(* CODESYS project xlh_palletizer_00_01.project
   Description: Receives some incoming messages and echoes them with CAN-ID +1
   Company: 3S - Smart Software Solutions GmbH
   Version: 1.0.0.0
   Title: CAN Bus API Example
   Author: 3S - Smart Software Solutions GmbH

Project tree, tasks and I/O mapping:
  xLH : CODESYS Control for Raspberry Pi 64 SL, CODESYS, order no. 2302000009, version 4.15.0.0
    application app
      libraries: Standard, 3.5.22.0 (System); Util, 3.5.22.0 (System); VisuDialogs, * (System); Memory, * (3S - Smart Software Solutions GmbH); xemax, 0.27 (xemax ag); CAN API, 1.0.0.4 (CODESYS)
      task MAIN_TASK (cyclic, interval 5 ms, priority 0) calls IO_READ, MAIN, MC, IO_WRITE
      task VISU_TASK (cyclic, interval 100 ms, priority 31) calls VisuElems.Visu_Prg
      task SoftMotion_PlanningTask (freewheeling, priority 15) calls nothing
      Symbols
      program MAIN [ST]
      visualisation Visualization
      MOTION/
        program MC [ST]: axSmExecuteToFalse, axGexecuteToFalse, axGenable, axGdisable, ipoGantry3
        trace PosControllerX (task MAIN_TASK): a1_axis.out.diSetVelocity, a1_axis.fSetAcceleration, a1_axis.fActPosition, a1_axis.fSetPosition, a1_axis.out.diSetVelocity
        function block FB_AXG_MOVE_ABSOLUTE [ST]
        function block FB_AXG_MOVE_RELATIVE [ST]
        trace PosController_A1_A2 (task MAIN_TASK): a1_axis.fSetPosition, a1_axis.fActPosition, a2_axis.fSetPosition, a2_axis.fActPosition
      IO/
        program IO_READ [ST]
        program io [ST]
        program IO_WRITE [ST]
      axis group AxisGroup: TRAFO.Kin_Gantry3, axes x_virtual, y_virtual, z_virtual
      text DemoInterpolator
      CNC settings
      text DemoXemaxLogo
      visualisation Visualization_1
      DOCS/
        Soft_Motion_Uebung_1_01_00
    SoftMotion General Axis Pool
      a3_axis : SM_Drive_PosControl, CODESYS, order no. 1805, version 4.18.0.0
          settings: wDriveID = 3; dwRatioTechUnitsDenom = 101846; iRatioTechUnitsNum = -125; eRampType = 0; fSWMaxAcceleration = 100; fSWMaxDeceleration = 100; fSWMaxJerk = 1000; fSWLimitNegative = -1000.0; ScalingIncs = 814768; ScalingUnits = 1000; InvertDirection = TRUE; IsLinearMotor = TRUE; MaximumOutputVelocityInt = 40738; MinimumOutputVelocityInt = -40738; Kp = 0.05; MaxFollowingError = 5.0; EnableFollowingErrorCheck = TRUE; DeadTime = 3.0
      a1_axis : SM_Drive_PosControl, CODESYS, order no. 1805, version 4.18.0.0
          settings: dwRatioTechUnitsDenom = 101846; iRatioTechUnitsNum = 125; eRampType = 0; fSWMaxVelocity = 50; fSWMaxAcceleration = 100; fSWMaxDeceleration = 100; fSWMaxJerk = 1000; fSWLimitNegative = -1000.0; ScalingIncs = 814768; ScalingUnits = 1000; IsLinearMotor = TRUE; MaximumOutputVelocityInt = 40738; MinimumOutputVelocityInt = -40738; Kp = 0.05; MaxFollowingError = 5.0; EnableFollowingErrorCheck = TRUE; DeadTime = 3.0
      a2_axis : SM_Drive_PosControl, CODESYS, order no. 1805, version 4.18.0.0
          settings: wDriveID = 2; dwRatioTechUnitsDenom = 101846; iRatioTechUnitsNum = 125; eRampType = 0; fSWMaxVelocity = 50; fSWMaxAcceleration = 100; fSWMaxDeceleration = 100; fSWMaxJerk = 1000; fSWLimitNegative = -1000.0; ScalingIncs = 814768; ScalingUnits = 1000; IsLinearMotor = TRUE; MaximumOutputVelocityInt = 40738; MinimumOutputVelocityInt = -40738; Kp = 0.05; MaxFollowingError = 5.0; EnableFollowingErrorCheck = TRUE; DeadTime = 3.0
      x_virtual : SM_Drive_Virtual, CODESYS, order no. 1805, version 4.18.0.0
          settings: wDriveID = 5; eRampType = 0; fSWMaxVelocity = 25; fSWMaxAcceleration = 100; fSWMaxDeceleration = 100; fSWMaxJerk = 1000; fSWLimitNegative = -1000.0
      y_virtual : SM_Drive_Virtual, CODESYS, order no. 1805, version 4.18.0.0
          settings: wDriveID = 6; eRampType = 0; fSWMaxVelocity = 25; fSWMaxAcceleration = 100; fSWMaxDeceleration = 100; fSWMaxJerk = 1000; fSWLimitNegative = -1000.0
      a4_axis : SM_Drive_PosControl, CODESYS, order no. 1805, version 4.18.0.0
          settings: wDriveID = 4; dwRatioTechUnitsDenom = 101846; iRatioTechUnitsNum = -125; eRampType = 0; fSWMaxAcceleration = 100; fSWMaxDeceleration = 100; fSWMaxJerk = 1000; fSWLimitNegative = -1000.0; ScalingIncs = 814768; ScalingUnits = 1000; InvertDirection = TRUE; IsLinearMotor = TRUE; MaximumOutputVelocityInt = 40738; MinimumOutputVelocityInt = -40738; Kp = 0.05; MaxFollowingError = 5.0; EnableFollowingErrorCheck = TRUE; DeadTime = 3.0
      z_virtual : SM_Drive_Virtual, CODESYS, order no. 1805, version 4.18.0.0
          settings: wDriveID = 7; eRampType = 0; fSWMaxVelocity = 25; fSWMaxAcceleration = 100; fSWMaxDeceleration = 100; fSWMaxJerk = 1000; fSWLimitNegative = -1000.0
    GPIOs_A_B : GPIOs B+/Pi2, CODESYS, version 4.15.0.0
        input  app.io.gpio.bSw1 : BOOL  // digital inputs (GPIO0..GPIO31).Bit4
        input  app.io.gpio.bSw2 : BOOL  // digital inputs (GPIO0..GPIO31).Bit5
        input  app.io.gpio.bSw3 : BOOL  // digital inputs (GPIO0..GPIO31).Bit6
        input  app.io.gpio.bSw4 : BOOL  // digital inputs (GPIO0..GPIO31).Bit12
        input  app.io.gpio.bSw5 : BOOL  // digital inputs (GPIO0..GPIO31).Bit13
        input  app.io.gpio.bSw6 : BOOL  // digital inputs (GPIO0..GPIO31).Bit16
        input  app.io.gpio.bSw7 : BOOL  // digital inputs (GPIO0..GPIO31).Bit17
        input  app.io.gpio.bSw8 : BOOL  // digital inputs (GPIO0..GPIO31).Bit19
        output app.io.gpio.bLed1 : BOOL  // digital outputs (GPIO0..GPIO31).Bit20
        output app.io.gpio.bLed2 : BOOL  // digital outputs (GPIO0..GPIO31).Bit21
        output app.io.gpio.bLed3 : BOOL  // digital outputs (GPIO0..GPIO31).Bit22
        output app.io.gpio.bLed4 : BOOL  // digital outputs (GPIO0..GPIO31).Bit23
        output app.io.gpio.bLed5 : BOOL  // digital outputs (GPIO0..GPIO31).Bit24
        output app.io.gpio.bLed6 : BOOL  // digital outputs (GPIO0..GPIO31).Bit26
        output app.io.gpio.bLed7 : BOOL  // digital outputs (GPIO0..GPIO31).Bit27
        unmapped channels: digital inputs (GPIO0..GPIO31), digital outputs (GPIO0..GPIO31)
    Onewire
    Camera device
      <Leer>
    SPI
    I²C
  libraries: VisuSymbols, 4.5.0.0 (System); DepictorBase, 1.2.0.0 (CODESYS)
  text list GlobalTextList
  00000000-0000-0000-0000-000000000000|E:\xemax ag\prj_24_03_xLH - Allgemein\Applikation\xLH_MOTION\CODESYS\Divers\080_SOFT_MOTION_PLC_OPEN\Soft_Motion_Uebung_1_01_00.pdf
*)

// xLH/app/IO/IO_READ
PROGRAM IO_READ
VAR
END_VAR

xemax.CAN_DRIVER();
io();
xemax.TASK_INFO();
xemax.LOCAL_TIME_AND_TIME_ZONE();

END_PROGRAM

// xLH/app/IO/io
PROGRAM io 
VAR_INPUT
	gpio: xemax.FB_XLH_GPIO;	
	motion: FB_XLH_MOTION := (uiCanIdBase:=16#300);
	xbox: FB_XBOX;
	bPenDown: BOOL;
END_VAR
VAR	
	bStartup: BOOL := TRUE;
	wdt: xemax.FB_XLH_WDT := (uiCanIdBase:=16#80);
	fbTonMagnet: TON;
END_VAR

IF bStartup THEN
	bStartup := FALSE;
	motion.pfbXlhMotionAxis[1] := ADR(MC.fbXlhMotionAxisA12.fbXlhMotionAxis1);
	motion.pfbXlhMotionAxis[2] := ADR(MC.fbXlhMotionAxisA12.fbXlhMotionAxis2);
	
	motion.uiIoOutPwmServo[9]  := 1000;
	
	CAN_DRIVER.mAddXlhDevice(pFbXlhIoDevice:=ADR(wdt));
	CAN_DRIVER.mAddXlhDevice(pFbXlhIoDevice:=ADR(motion));	
END_IF

xbox();

(*
IF io.bPenDown OR (z_virtual.fActPosition < (-1.0)) THEN
	motion.uiIoOutPwmServo[9]  := 1200;
ELSE
	motion.uiIoOutPwmServo[9]  := 800;
END_IF
*)

IF MC.iState < 3000 THEN
	IF bPenDown THEN
		motion.uiIoOutPwmServo[9]  := 1200;
	ELSE
		motion.uiIoOutPwmServo[9]  := 800;
	END_IF
ELSE
	IF z_virtual.fActPosition < (-1.0) THEN
		motion.uiIoOutPwmServo[9]  := 1200;
	ELSE
		motion.uiIoOutPwmServo[9]  := 800;
	END_IF
END_IF

END_PROGRAM

// xLH/app/MOTION/MC
PROGRAM MC
VAR_OUTPUT
	iState: INT;	
END_VAR
VAR
	bStartup: BOOL := TRUE;
	fbBlink: BLINK;
	
	axA1: FB_PLC_OPEN_AXIS := (rVel:=VEL, rAcc:=ACC_DEC, rDec:=ACC_DEC, rJerk:=JRK);
	axA2: FB_PLC_OPEN_AXIS := (rVel:=VEL, rAcc:=ACC_DEC, rDec:=ACC_DEC, rJerk:=JRK);
	axVx: FB_PLC_OPEN_AXIS := (rVel:=VEL, rAcc:=ACC_DEC, rDec:=ACC_DEC, rJerk:=JRK);
	axVy: FB_PLC_OPEN_AXIS := (rVel:=VEL, rAcc:=ACC_DEC, rDec:=ACC_DEC, rJerk:=JRK);
	axVz: FB_PLC_OPEN_AXIS := (rVel:=VEL, rAcc:=ACC_DEC, rDec:=ACC_DEC, rJerk:=JRK);
	fbXlhMotionAxisA12: FB_XLH_MOTION_AXIS_MID_T_BOT;
	fbTonDelay1: TON := (PT := TIME#1S0MS);
	fbTonDelay2: TON := (PT := TIME#1S0MS);	
	
	mcAxGenable : MC_GroupEnable;
	mcAxGdisable : MC_GroupDisable;
	mcAxGreset: MC_GroupReset;
	mcAxGsetCoord : MC_SetCoordinateTransform;	
	mcAxGmla: MC_MoveLinearAbsolute := (Velocity := VEL, Acceleration := ACC_DEC, Deceleration := ACC_DEC, Jerk := JRK);
	mcAxGmlr: MC_MoveLinearRelative := (Velocity := VEL, Acceleration := ACC_DEC, Deceleration := ACC_DEC, Jerk := JRK);	
	mcAxGcoordRef : MC_COORD_REF;
	smcPosRef: SMC_POS_REF;
	
	fbAxGmr: FB_AXG_MOVE_RELATIVE;
	fbAxGma: FB_AXG_MOVE_ABSOLUTE;
	
	rStepDistance: REAL := 15.0;
	rStpNeg: REAL;
	rStpPos: REAL;
	
	tPosMC : SMC_POS_REF ;
	smcGroupReadSetPosition : SMC_GroupReadSetPosition := (Enable:= TRUE, CoordSystem:= SMC_COORD_SYSTEM.MCS) ;
	mcGroupReadStatus: MC_GroupReadStatus;
	
	smcControlAxByPosA1: SMC_ControlAxisByPos;
	smcControlAxByPosA2: SMC_ControlAxisByPos;

	smcTrafoGantry3d: SMC_TRAFO_Gantry3;
	smcTrafofGantry3d: SMC_TRAFOF_Gantry3D;
	smcControlAxByPosX,smcControlAxByPosY, smcControlAxByPosZ: SMC_ControlAxisByPos;
	smcInterpolator: SMC_Interpolator;
	
	rOffsetX: REAL := 0.0;
	rOffsetY: REAL := -10.0;
	
	bVisuXplus: BOOL;
	bVisuXminus: BOOL;
	bVisuYplus: BOOL;
	bVisuYminus: BOOL;
	bVisuPenDown: BOOL;
	bVisuStartNc: BOOL;
	bVisuHoming: BOOL;
	
END_VAR
VAR CONSTANT
	VEL : REAL := 15.0;
	VEL_HOMING : REAL := 2.0;
    ACC_DEC : REAL := 100.0;
    JRK : REAL := 1000.0;	
END_VAR
VAR // added by the converter: edge detectors and wires of the graphical bodies
    _w1 : ANY;
END_VAR

// ToDo: Optimierung
IF bStartup THEN
	bStartup := FALSE;
	axA1.pAxis := ADR(a1_axis);
	axA2.pAxis := ADR(a2_axis);
	axVx.pAxis := ADR(x_virtual);
	axVy.pAxis := ADR(y_virtual);
	axVz.pAxis := ADR(z_virtual);
	
	fbXlhMotionAxisA12.fbXlhMotionAxis1.pAxis := ADR(a1_axis);
	fbXlhMotionAxisA12.fbXlhMotionAxis2.pAxis := ADR(a2_axis);
	fbXlhMotionAxisA12.pfbAxisPlcOpenX := ADR(axVx);
	fbXlhMotionAxisA12.pfbAxisPlcOpenY := ADR(axVy);
	fbXlhMotionAxisA12.pbEsX := ADR(io.motion.bIoIn[5]);
	fbXlhMotionAxisA12.pbEsY := ADR(io.motion.bIoIn[1]);
	
	fbAxGmr.axGmr REF= mcAxGmlr;
	fbAxGmr.axG REF= AxisGroup;  
	fbAxGma.axGma REF= mcAxGmla;
	fbAxGma.axG REF= AxisGroup;
	fbAxGma.axG REF= AxisGroup;
END_IF

axA1();
axA2();
fbXlhMotionAxisA12();
axVx();
axVy();
axVz();
MC.ipoGantry3();

// ToDo: Optimierung
mcAxGmla(AxisGroup:= AxisGroup);
mcAxGmlr(AxisGroup:= AxisGroup);
fbAxGmr();
fbAxGma();
mcGroupReadStatus(Enable:=TRUE, AxisGroup:=AxisGroup);
smcGroupReadSetPosition(Enable:=TRUE, AxisGroup:=AxisGroup, Position=>tPosMC);

tPosMC.c.X;
tPosMC.c.Y;
tPosMC.c.Z;
tPosMC.c.A;
tPosMC.c.B;
tPosMC.c.C;
a1_axis.fActPosition;
a2_axis.fActPosition;
x_virtual.fActPosition;
y_virtual.fActPosition;
z_virtual.fActPosition;

// kinematische Transformation
smcControlAxByPosA1(Axis:=a1_axis,
	        bEnable:= (iState >= 100),
            iStatus:=IPO_WAIT,
		    fSetPosition:= (+2.0) * x_virtual.fSetPosition + (+1.0) * y_virtual.fSetPosition,
			fGapVelocity:=VEL,
            fGapAcceleration:=ACC_DEC,
            fGapDeceleration:=ACC_DEC);
smcControlAxByPosA2(Axis:=a2_axis,
	        bEnable:= (iState >= 100),
            iStatus:=IPO_WAIT,
		    fSetPosition:= (+2.0) * x_virtual.fSetPosition - (+1.0) * y_virtual.fSetPosition,
			fGapVelocity:=VEL,
            fGapAcceleration:=ACC_DEC,
            fGapDeceleration:=ACC_DEC);

CASE iState OF
	// ============================================================================================
	// STARTUP UND INITIALISIERUNG
	// ============================================================================================
	
	0:		// Startup
			MC.axSmExecuteToFalse();
			MC.axGexecuteToFalse();		
			iState := 50;
			
	50:	// Power der Achsen
			axA1.mcp.Enable := TRUE; axA1.mcp.bRegulatorOn := TRUE; axA1.mcp.bDriveStart := TRUE;
			axA2.mcp.Enable := TRUE; axA2.mcp.bRegulatorOn := TRUE; axA2.mcp.bDriveStart := TRUE;
			// https://content.helpme-codesys.com/en/libs/SM3_Basic/Current/SM3_Basic/DataTypes/DriveInterface/SMC_AXIS_STATE.html
			IF (axA1.mcp.Status AND a1_axis.nAxisState = SMC_AXIS_STATE.standstill) AND
	           (axA2.mcp.Status AND a2_axis.nAxisState = SMC_AXIS_STATE.standstill) THEN
				MC.axSmExecuteToFalse();
				iState := iState + 10;
			END_IF
			
	60: // Power der Achsen
		axVx.mcp.Enable := TRUE; axVx.mcp.bRegulatorOn := TRUE; axVx.mcp.bDriveStart := TRUE;
		axVy.mcp.Enable := TRUE; axVy.mcp.bRegulatorOn := TRUE; axVy.mcp.bDriveStart := TRUE;
		axVz.mcp.Enable := TRUE; axVz.mcp.bRegulatorOn := TRUE; axVz.mcp.bDriveStart := TRUE;
		// https://content.helpme-codesys.com/en/libs/SM3_Basic/Current/SM3_Basic/DataTypes/DriveInterface/SMC_AXIS_STATE.html
		IF (axVx.mcp.Status AND x_virtual.nAxisState = SMC_AXIS_STATE.standstill) AND
		   (axVy.mcp.Status AND y_virtual.nAxisState = SMC_AXIS_STATE.standstill) AND
           (axVz.mcp.Status AND z_virtual.nAxisState = SMC_AXIS_STATE.standstill) THEN
			MC.axSmExecuteToFalse();
			iState := iState + 10;
		END_IF
		
	70: 	iState := 100;

	100:	// Disable der Achsengruppe		
			IF NOT mcGroupReadStatus.GroupDisabled THEN
				mcAxGdisable(AxisGroup := AxisGroup, Execute := TRUE);	
				IF mcAxGdisable.Done THEN
					MC.axGexecuteToFalse();
					iState := iState + 10;
				END_IF
			ELSE
				iState := iState + 10;
			END_IF	
			
	//110:	iState := iState + 20;

	110:	// Homing
			fbXlhMotionAxisA12.bHoming := TRUE;
			fbXlhMotionAxisA12.rVelHoming := VEL_HOMING;
			fbXlhMotionAxisA12.rVelHomingFast := 5.0 * VEL_HOMING;
			fbXlhMotionAxisA12.rOffsetX := 38.0;
			fbXlhMotionAxisA12.rOffsetY := -40.0;
			
			axVz.mcma.Execute := TRUE;
			axVz.mcma.Position := 0.0;
			axVz.mcma.Velocity := z_virtual.fSWMaxVelocity;
			
			IF fbXlhMotionAxisA12.bHomingDone AND
               axVz.mcma.Done THEN
				MC.axSmExecuteToFalse();
				fbXlhMotionAxisA12.bHoming := FALSE;
				iState := iState + 10;
			END_IF	
		
	120: 	iState := 1000;
	
	// ============================================================================================
	// Kommandos
	// ============================================================================================
	
	1000: 	// Resetierung der Kommandos
			MC.axSmExecuteToFalse();
			MC.axGexecuteToFalse();		
			
			bVisuXplus := FALSE;
			bVisuXminus := FALSE;
			bVisuYplus := FALSE;
			bVisuYminus := FALSE;
			//bVisuPenDown := FALSE;
			bVisuStartNc := FALSE;
			bVisuHoming := FALSE;
			
			iState := iState + 10;
			
	1010:	// warte auf Aktion					
			IF io.xbox.bRtBtnRightShoulder OR bVisuHoming THEN iState := 100; END_IF
						
			rStpNeg := rStepDistance * (-1.0);
			rStpPos := rStepDistance;
			
			IF io.xbox.bBtnB OR bVisuXplus    THEN smcPosRef.c.X := rStpPos; smcPosRef.c.Y := 0.0;	    iState := 2000; END_IF
			IF io.xbox.bBtnX OR bVisuXminus   THEN smcPosRef.c.X := rStpNeg; smcPosRef.c.Y := 0.0;	    iState := 2000; END_IF
			IF io.xbox.bBtnY OR bVisuYplus    THEN smcPosRef.c.X := 0.0;     smcPosRef.c.Y := rStpPos;	iState := 2000; END_IF
			IF io.xbox.bBtnA OR bVisuYminus   THEN smcPosRef.c.X := 0.0;     smcPosRef.c.Y := rStpNeg;	iState := 2000; END_IF
					
			//IF io.xbox.bBtnDpadUp   THEN io.bPenDown := FALSE; END_IF
			//IF io.xbox.bBtnDpadDown THEN io.bPenDown := TRUE;  END_IF
			io.bPenDown := bVisuPenDown;

			IF io.xbox.bBtnStart OR bVisuStartNc THEN iState := 3000; END_IF  
			
	// ============================================================================================
	// Stepbetrieb der Achsen
	// ============================================================================================
	
	// ToDo: Optimierung und Abstrahierung als FB
	
	
	2000:	MC.axGenable();
	2001: 	smcPosRef.c.Z := 0.0;
			fbAxGmr.bExecute := TRUE;
			fbAxGmr.tPosRef := smcPosRef;
			IF fbAxGmr.bDone THEN
				MC.axGexecuteToFalse();
				iState := iState + 1;
			END_IF
	2002:	MC.axGdisable();
	2003:	iState := 1000;
	
	2010:	MC.axGenable();
	2011: 	smcPosRef.c.Z := tPosMC.c.Z;
			fbAxGma.bExecute := TRUE;
			fbAxGma.tPosRef := smcPosRef;
			IF fbAxGma.bDone THEN
				MC.axGexecuteToFalse();
				iState := 1000;
			END_IF
	2012:	MC.axGdisable();
	2013:	iState := 1000;
			
	
	(*		
	2020: 	// Stifthalterung 
			smcPosRef.c.X := tPosMC.c.X;
			smcPosRef.c.Y := tPosMC.c.Y;
			IF io.bPenDown THEN
				smcPosRef.c.Z := -10.0;
			ELSE
				smcPosRef.c.Z := 0.0;
			END_IF
			fbAxGma.bExecute := TRUE;
			fbAxGma.tPosRef := smcPosRef;
			IF fbAxGma.bDone THEN
				MC.axGexecuteToFalse();
				iState := 1000;
			END_IF
	*)
	
	// ============================================================================================
	// Interpolator
	// ============================================================================================
	
	3000:	bVisuPenDown := FALSE;
			axVx.mcma.Execute := TRUE;
			axVx.mcma.Position := rOffsetX;
			axVy.mcma.Execute := TRUE;
			axVy.mcma.Position := rOffsetY;
			axVz.mcma.Execute := TRUE;
			axVz.mcma.Position := 0.0;
			IF axVx.mcma.Done AND axVy.mcma.Done AND axVz.mcma.Done THEN
				MC.axSmExecuteToFalse();
				iState := iState + 10;
			END_IF
			
	3010:	smcInterpolator.bExecute := TRUE;
			IF smcInterpolator.bDone THEN
				MC.axSmExecuteToFalse();
				iState := iState + 10;
			END_IF
			
	3020:	axVx.mcma.Execute := TRUE;
			axVx.mcma.Position := 0.0;
			axVy.mcma.Execute := TRUE;
			axVy.mcma.Position := 0.0;
			axVz.mcma.Execute := TRUE;
			axVz.mcma.Position := 0.0;
			IF axVx.mcma.Done AND axVy.mcma.Done AND axVz.mcma.Done THEN
				MC.axSmExecuteToFalse();
				iState := iState + 10;
			END_IF
	
	3030: 	iState := 1000;
	
	
END_CASE

fbTonDelay1();
fbTonDelay2();
fbTonDelay1.IN := FALSE;
fbTonDelay2.IN := FALSE;

ACTION axSmExecuteToFalse:
axA1.executeToFalse();
axA2.executeToFalse();
axVx.executeToFalse();
axVy.executeToFalse();
axVz.executeToFalse();

smcInterpolator.bExecute := FALSE;
END_ACTION

ACTION axGexecuteToFalse:
mcAxGenable(AxisGroup := AxisGroup, Execute := FALSE);
mcAxGdisable(AxisGroup := AxisGroup, Execute := FALSE);
mcAxGreset(AxisGroup := AxisGroup, Execute := FALSE);
mcAxGsetCoord(AxisGroup := AxisGroup, Execute := FALSE);

fbAxGma.bExecute := FALSE;
fbAxGmr.bExecute := FALSE;
mcAxGmla(AxisGroup := AxisGroup, Execute := FALSE);
mcAxGmlr(AxisGroup := AxisGroup, Execute := FALSE);
END_ACTION

ACTION axGenable:
// Enable der Achsengruppe
IF mcGroupReadStatus.GroupDisabled THEN 
	mcAxGenable(AxisGroup := AxisGroup, Execute := TRUE);	
	IF mcAxGenable.Done THEN
		MC.axGexecuteToFalse();
		iState := iState + 1;
		//iState := 580;
	END_IF			
END_IF	

// ToDo: Verallgemeinerung und Auslagerung in FB
END_ACTION

ACTION axGdisable:
// Disable der Achsengruppe		
IF NOT mcGroupReadStatus.GroupDisabled THEN
	mcAxGdisable(AxisGroup := AxisGroup, Execute := TRUE);	
	IF mcAxGdisable.Done THEN
		MC.axGexecuteToFalse();
		iState := iState + 1;
	END_IF
END_IF

// ToDo: Verallgemeinerung und Auslagerung in FB
END_ACTION

ACTION ipoGantry3:
smcTrafofGantry3d(
    minX := -50.0,
    maxX := 50.0,
    minY := -50.0,
    maxY := 50.0,
    minZ := -10.0,
    maxZ := 0.0,
    DriveX := x_virtual,
    DriveY := y_virtual,
    DriveZ := z_virtual); // SMC_TRAFOF_Gantry3D
smcControlAxByPosX(
    iStatus := smcInterpolator.iStatus,
    bEnable := smcInterpolator.bWorking,
    fSetPosition := smcTrafoGantry3d.dx,
    fGapVelocity := 10.0,
    fGapAcceleration := 100.0,
    fGapDeceleration := 100.0,
    Axis := x_virtual); // SMC_ControlAxisByPos
smcInterpolator(poqDataIn := ADR(DemoInterpolator), bEmergency_Stop := _w1, dwIpoTime := 5000); // SMC_Interpolator
smcTrafoGantry3d(pi := smcInterpolator.piSetPosition, dOffsetX := rOffsetX, dOffsetY := rOffsetY); // SMC_TRAFO_Gantry3
smcControlAxByPosY(
    iStatus := smcInterpolator.iStatus,
    bEnable := smcInterpolator.bWorking,
    fSetPosition := smcTrafoGantry3d.dy,
    fGapVelocity := 10.0,
    fGapAcceleration := 100.0,
    fGapDeceleration := 100.0,
    Axis := y_virtual); // SMC_ControlAxisByPos
smcControlAxByPosZ(
    iStatus := smcInterpolator.iStatus,
    bEnable := smcInterpolator.bWorking,
    fSetPosition := smcTrafoGantry3d.dz,
    fGapVelocity := 10.0,
    fGapAcceleration := 100.0,
    fGapDeceleration := 100.0,
    Axis := z_virtual); // SMC_ControlAxisByPos
_w1 := smcControlAxByPosX.bError OR smcControlAxByPosX.bStopIpo OR smcControlAxByPosY.bError OR smcControlAxByPosY.bStopIpo OR smcControlAxByPosZ.bError OR smcControlAxByPosZ.bStopIpo;
END_ACTION

END_PROGRAM

// xLH/app/MOTION/FB_AXG_MOVE_RELATIVE
FUNCTION_BLOCK FB_AXG_MOVE_RELATIVE
VAR_INPUT
	bExecute: BOOL;
	tPosRef: SMC_POS_REF;
	axGmr: REFERENCE TO MC_MoveLinearRelative;
	axG: REFERENCE TO AXIS_GROUP_REF_SM3;
END_VAR
VAR_OUTPUT
	bDone: BOOL;
END_VAR

axGmr.Execute := bExecute;
axGmr.Distance := tPosRef;
axGmr.BufferMode := MC_BUFFER_MODE.BlendingHigh;
axGmr.TransitionMode := MC_TRANSITION_MODE.TMCornerDistance;
axGmr.TransitionParameter[0] := 50;
//axGmvTo.CoordSystem := SMC_COORD_SYSTEM.PCS_1;
axGmr.CoordSystem := SMC_COORD_SYSTEM.MCS;
bDone := axGmr.Done;

END_FUNCTION_BLOCK

// xLH/app/MOTION/FB_AXG_MOVE_ABSOLUTE
FUNCTION_BLOCK FB_AXG_MOVE_ABSOLUTE
VAR_INPUT
	bExecute: BOOL;
	tPosRef: SMC_POS_REF;
	axGma: REFERENCE TO MC_MoveLinearAbsolute;
	axG: REFERENCE TO AXIS_GROUP_REF_SM3;
END_VAR
VAR_OUTPUT
	bDone: BOOL;
END_VAR

axGma.Execute := bExecute;
axGma.Position := tPosRef;
axGma.BufferMode := MC_BUFFER_MODE.BlendingHigh;
axGma.TransitionMode := MC_TRANSITION_MODE.TMCornerDistance;
axGma.TransitionParameter[0] := 50;
//axGmvTo.CoordSystem := SMC_COORD_SYSTEM.PCS_1;
axGma.CoordSystem := SMC_COORD_SYSTEM.MCS;
bDone := axGma.Done;

END_FUNCTION_BLOCK

// xLH/app/MAIN
PROGRAM MAIN
VAR
	vVersionPlc: VERSION;
	sVersionPlc: STRING(255);
	vVersionLib: VERSION;
	sVersionLib: STRING(255);
	bStartup: BOOL := TRUE;

	bSimulation: BOOL;
	iCtr: INT;
END_VAR

// Version Bibliothex xemax
vVersionPlc.uiMajor := 1;
vVersionPlc.uiMinor := 0;
sVersionPlc := CONCAT(TO_STRING(TO_UINT(vVersionPlc.uiMajor)), CONCAT('.', (TO_STRING(TO_UINT(vVersionPlc.uiMinor)))));
vVersionLib := xemax.GetLibVersion();
sVersionLib := CONCAT(TO_STRING(TO_UINT(vVersionLib.uiMajor)), CONCAT('.', (TO_STRING(TO_UINT(vVersionLib.uiMinor)))));

IF bStartup THEN
	bStartup := FALSE;

END_IF


// Erkennung Simulationsmodus
// https://content.helpme-codesys.com/en/LibDevSummary/friends.html
bSimulation := __SYSTEM.Constants.bSimulationMode;

{IF NOT defined (IsSimulationMode)}
	iCtr := iCtr + 1;
{ELSE}
	iCtr := iCtr - 1;
{END_IF}

END_PROGRAM

// xLH/app/IO/IO_WRITE
PROGRAM IO_WRITE
VAR
	fbTofSm1: TOF;
END_VAR

xemax.CAN_DRIVER.mWrite();

END_PROGRAM

// xLH/app/Visualization
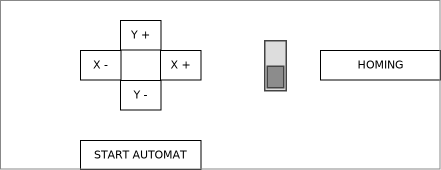
VISUALIZATION Visualization  // 441x170
    Rectangle (120,20 41x30), "Y +"
        toggle MC.bVisuYplus
    Rectangle (120,80 41x30), "Y -"
        toggle MC.bVisuYminus
    Rectangle (80,50 41x30), "X -"
        toggle MC.bVisuXminus
    Rectangle (160,50 41x30), "X +"
        toggle MC.bVisuXplus
    DipSwitch (250,40 51x51), variable: MC.bVisuPenDown, behaviour: TOGGLE, style: Switch-DipSwitch-Gray
    Rectangle (80,140 121x30), "START AUTOMAT"
        toggle MC.bVisuStartNc
    Rectangle (320,50 121x30), "HOMING"
        toggle MC.bVisuHoming
END_VISUALIZATION

// xLH/app/Visualization_1
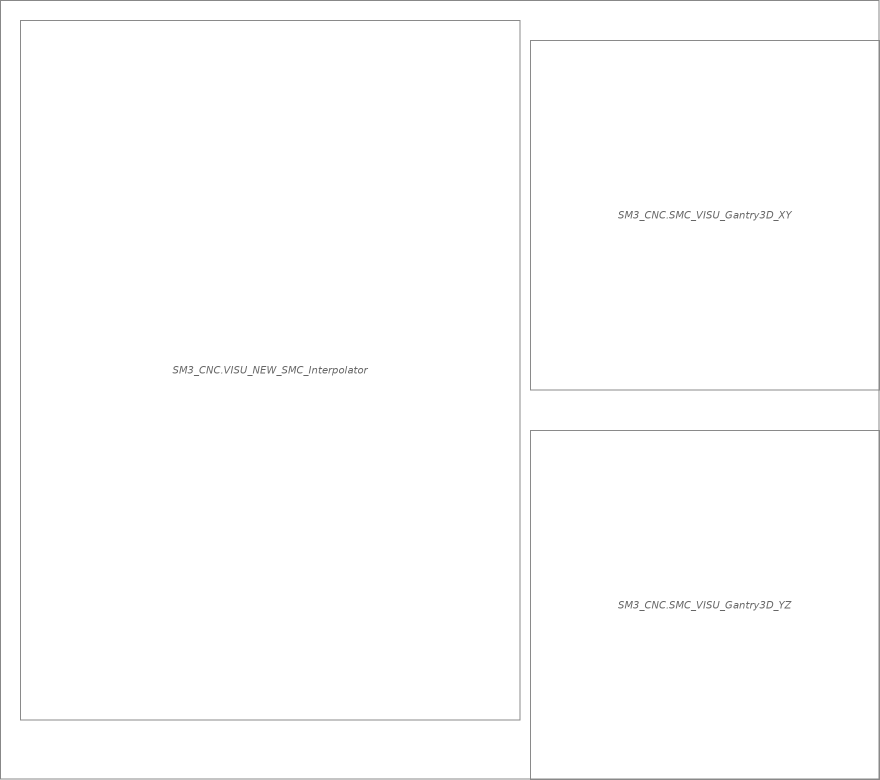
VISUALIZATION Visualization_1  // 880x780
    Frame (20,20 500x700)
        shows SM3_CNC.VISU_NEW_SMC_Interpolator(m_Input_FB := MC.smcInterpolator)
    Frame (530,430 350x350)
        shows SM3_CNC.SMC_VISU_Gantry3D_YZ(m_Input_SMC_TrafoF_Gantry := MC.smcTrafofGantry3d)
    Frame (530,40 350x350)
        shows SM3_CNC.SMC_VISU_Gantry3D_XY(m_Input_SMC_TrafoF_Gantry := MC.smcTrafofGantry3d)
END_VISUALIZATION

(* text DemoInterpolator
N000 G01 X0 Y0 Z0 E100 E-100 F15
N010 G00 X-25 Y0 
N020 G01 Z-5.0 
N030 G01 X-25 Y22.5 
N040 G02 X-22.5 Y25 I2.5 J0 
N050 G01 X-15 Y25 
N060 G02 X15 Y25 I15 J0 K180 
N070 G01 X22.5 Y25 
N080 G02 X25 Y22.5 I0 J-2.5 
N090 G01 X25 Y0 
N100 G01 X-25 Y0 
N110 G00 Z10 
N120 G00 X-11.25 Y12.5 
N130 G00 Z-10.0 
N140 G02 I-5 J0 
N150 G00 Z10 
N160 G00 X11.25 Y12.5 
N170 G00 Z-10.0 
N180 G02 I5 J0
N190 G00 Z10 
N200 G00 X0 Y0
*)

(* text DemoXemaxLogo
N000 G01 X0 Y0 Z0 E100 E-100 F15 
N010 G00 X0.007 Y-2.042 Z5 
N020 G01 Z-5 F254 
N030 G01 X0.067 F1200 
N040 X0.125 
N050 X0.183 
N060 X0.241 
N070 X0.297 
N080 X0.353 
N090 X0.409 
N100 X0.464 
N110 X0.518 
N120 X0.571 
N130 X0.624 
N140 X0.676 
N150 X0.727 
N160 X0.778 
N170 X0.828 
N180 X0.877 
N190 X0.925 
N200 X0.973 
N210 X1.019 
N220 X1.065 
N230 X1.11 
N240 X1.155 
N250 X1.198 
N260 X1.241 
N270 X1.282 
N280 X1.323 
N290 X1.363 
N300 X1.402 
N310 X1.44 
N320 X1.478 
N330 X1.514 
N340 X1.549 
N350 X1.584 
N360 X1.617 
N370 X1.65 
N380 X1.681 
N390 X1.712 
N400 X1.741 
N410 X1.77 
N420 X1.797 
N430 X1.824 
N440 X1.849 
N450 X1.873 
N460 X1.896 
N470 X1.919 
N480 X1.94 
N490 X1.959 
N500 X1.978 
N510 X1.996 
N520 X2.012 
N530 X2.028 
N540 X2.042 
N550 X2.055 
N560 X2.066 
N570 X2.077 
N580 X2.086 
N590 X2.095 
N600 X2.101 
N610 X2.107 
N620 X2.111 
N630 X2.114 
N640 X2.116 
N650 X2.117 Y-2.042 
N660 X2.117 Y-2.043 
N670 X2.118 Y-2.044 
N680 X2.119 Y-2.045 
N690 X2.121 Y-2.047 
N700 X2.124 Y-2.049 
N710 X2.127 Y-2.052 
N720 X2.13 Y-2.056 
N730 X2.134 Y-2.06 
N740 X2.139 Y-2.065 
N750 X2.144 Y-2.07 
N760 X2.15 Y-2.075 
N770 X2.156 Y-2.081 
N780 X2.162 Y-2.088 
N790 X2.169 Y-2.095 
N800 X2.177 Y-2.102 
N810 X2.185 Y-2.11 
N820 X2.193 Y-2.119 
N830 X2.202 Y-2.128 
N840 X2.211 Y-2.137 
N850 X2.221 Y-2.147 
N860 X2.232 Y-2.157 
N870 X2.242 Y-2.168 
N880 X2.253 Y-2.179 
N890 X2.265 Y-2.191 
N900 X2.277 Y-2.203 
N910 X2.29 Y-2.215 
N920 X2.302 Y-2.228 
N930 X2.316 Y-2.241 
N940 X2.33 Y-2.255 
N950 X2.344 Y-2.269 
N960 X2.358 Y-2.284 
N970 X2.373 Y-2.299 
N980 X2.388 Y-2.314 
N990 X2.404 Y-2.33 
N1000 X2.42 Y-2.346 
N1010 X2.437 Y-2.362 
N1020 X2.454 Y-2.379 
N1030 X2.471 Y-2.396 
N1040 X2.488 Y-2.414 
N1050 X2.506 Y-2.432 
N1060 X2.525 Y-2.45 
N1070 X2.543 Y-2.469 
N1080 X2.562 Y-2.488 
N1090 X2.582 Y-2.507 
N1100 X2.601 Y-2.527 
N1110 X2.621 Y-2.547 
N1120 X2.642 Y-2.567 
N1130 X2.662 Y-2.588 
N1140 X2.683 Y-2.609 
N1150 X2.726 Y-2.652 
N1160 X2.77 Y-2.696 
N1170 X2.816 Y-2.741 
N1180 X2.862 Y-2.788 
N1190 X2.91 Y-2.835 
N1200 X2.958 Y-2.884 
N1210 X3.008 Y-2.933 
N1220 X3.058 Y-2.984 
N1230 X3.11 Y-3.035 
N1240 X3.162 Y-3.088 
N1250 X3.215 Y-3.141 
N1260 X3.269 Y-3.195 
N1270 X3.324 Y-3.25 
N1280 X3.38 Y-3.305 
N1290 X3.436 Y-3.362 
N1300 X3.493 Y-3.419 
N1310 X3.551 Y-3.476 
N1320 X3.609 Y-3.534 
N1330 X3.668 Y-3.593 
N1340 X3.727 Y-3.653 
N1350 X3.787 Y-3.712 
N1360 X3.847 Y-3.772 
N1370 X3.907 Y-3.833 
N1380 X3.968 Y-3.894 
N1390 X4.03 Y-3.955 
N1400 X4.153 Y-4.079 
N1410 X4.277 Y-4.203 
N1420 X4.402 Y-4.327 
N1430 X4.651 Y-4.577 
N1440 X4.776 Y-4.701 
N1450 X4.899 Y-4.825 
N1460 X5.022 Y-4.948 
N1470 X5.083 Y-5.008 
N1480 X5.143 Y-5.069 
N1490 X5.203 Y-5.129 
N1500 X5.263 Y-5.188 
N1510 X5.322 Y-5.248 
N1520 X5.38 Y-5.306 
N1530 X5.438 Y-5.364 
N1540 X5.496 Y-5.421 
N1550 X5.553 Y-5.478 
N1560 X5.609 Y-5.534 
N1570 X5.664 Y-5.59 
N1580 X5.719 Y-5.644 
N1590 X5.772 Y-5.698 
N1600 X5.825 Y-5.751 
N1610 X5.877 Y-5.803 
N1620 X5.929 Y-5.854 
N1630 X5.979 Y-5.904 
N1640 X6.028 Y-5.954 
N1650 X6.076 Y-6.002 
N1660 X6.123 Y-6.049 
N1670 X6.169 Y-6.095 
N1680 X6.214 Y-6.14 
N1690 X6.258 Y-6.184 
N1700 X6.301 Y-6.226 
N1710 X6.321 Y-6.247 
N1720 X6.342 Y-6.267 
N1730 X6.362 Y-6.287 
N1740 X6.382 Y-6.307 
N1750 X6.401 Y-6.327 
N1760 X6.42 Y-6.346 
N1770 X6.439 Y-6.365 
N1780 X6.457 Y-6.383 
N1790 X6.476 Y-6.401 
N1800 X6.493 Y-6.419 
N1810 X6.511 Y-6.436 
N1820 X6.528 Y-6.453 
N1830 X6.544 Y-6.47 
N1840 X6.56 Y-6.486 
N1850 X6.576 Y-6.502 
N1860 X6.592 Y-6.517 
N1870 X6.607 Y-6.532 
N1880 X6.621 Y-6.547 
N1890 X6.636 Y-6.561 
N1900 X6.65 Y-6.575 
N1910 X6.663 Y-6.589 
N1920 X6.676 Y-6.602 
N1930 X6.689 Y-6.614 
N1940 X6.701 Y-6.626 
N1950 X6.713 Y-6.638 
N1960 X6.724 Y-6.65 
N1970 X6.735 Y-6.66 
N1980 X6.745 Y-6.671 
N1990 X6.755 Y-6.681 
N2000 X6.765 Y-6.69 
N2010 X6.774 Y-6.699 
N2020 X6.782 Y-6.708 
N2030 X6.791 Y-6.716 
N2040 X6.798 Y-6.724 
N2050 X6.805 Y-6.731 
N2060 X6.812 Y-6.738 
N2070 X6.818 Y-6.744 
N2080 X6.824 Y-6.75 
N2090 X6.829 Y-6.755 
N2100 X6.834 Y-6.76 
N2110 X6.838 Y-6.764 
N2120 X6.842 Y-6.768 
N2130 X6.845 Y-6.771 
N2140 X6.848 Y-6.773 
N2150 X6.85 Y-6.775 
N2160 X6.851 Y-6.777 
N2170 X6.853 Y-6.778 
N2180 X6.853 Y-6.779 
N2190 X6.853 Y-6.781 
N2200 Y-6.785 
N2210 Y-6.791 
N2220 Y-6.798 
N2230 Y-6.807 
N2240 Y-6.817 
N2250 Y-6.829 
N2260 Y-6.842 
N2270 Y-6.857 
N2280 Y-6.873 
N2290 Y-6.89 
N2300 Y-6.909 
N2310 Y-6.93 
N2320 Y-6.951 
N2330 Y-6.974 
N2340 Y-6.998 
N2350 Y-7.024 
N2360 Y-7.05 
N2370 Y-7.078 
N2380 Y-7.107 
N2390 Y-7.137 
N2400 Y-7.168 
N2410 Y-7.2 
N2420 Y-7.233 
N2430 Y-7.267 
N2440 Y-7.302 
N2450 Y-7.337 
N2460 Y-7.374 
N2470 Y-7.412 
N2480 Y-7.45 
N2490 Y-7.489 
N2500 Y-7.529 
N2510 Y-7.57 
N2520 Y-7.612 
N2530 Y-7.654 
N2540 Y-7.696 
N2550 Y-7.74 
N2560 Y-7.784 
N2570 Y-7.828 
N2580 Y-7.873 
N2590 Y-7.919 
N2600 Y-8.011 
N2610 Y-8.105 
N2620 Y-8.2 
N2630 Y-8.297 
N2640 Y-8.394 
N2650 Y-8.492 
N2660 Y-8.688 
N2670 Y-8.884 
N2680 Y-8.982 
N2690 Y-9.078 
N2700 Y-9.174 
N2710 Y-9.268 
N2720 Y-9.36 
N2730 Y-9.406 
N2740 Y-9.451 
N2750 Y-9.496 
N2760 Y-9.54 
N2770 Y-9.583 
N2780 Y-9.626 
N2790 Y-9.668 
N2800 Y-9.71 
N2810 Y-9.751 
N2820 Y-9.791 
N2830 Y-9.83 
N2840 Y-9.869 
N2850 Y-9.907 
N2860 Y-9.944 
N2870 Y-9.98 
N2880 Y-10.015 
N2890 Y-10.049 
N2900 Y-10.082 
N2910 Y-10.115 
N2920 Y-10.146 
N2930 Y-10.176 
N2940 Y-10.205 
N2950 Y-10.233 
N2960 Y-10.26 
N2970 Y-10.285 
N2980 Y-10.31 
N2990 Y-10.333 
N3000 Y-10.355 
N3010 Y-10.375 
N3020 Y-10.395 
N3030 Y-10.412 
N3040 Y-10.429 
N3050 Y-10.444 
N3060 Y-10.458 
N3070 Y-10.47 
N3080 Y-10.48 
N3090 Y-10.489 
N3100 Y-10.497 
N3110 Y-10.503 
N3120 Y-10.507 
N3130 Y-10.509 
N3140 Y-10.51 
N3150 X6.882 Y-10.525 
N3160 X6.911 Y-10.541 
N3170 X6.94 Y-10.557 
N3180 X6.968 Y-10.574 
N3190 X6.996 Y-10.591 
N3200 X7.024 Y-10.608 
N3210 X7.051 Y-10.626 
N3220 X7.078 Y-10.645 
N3230 X7.105 Y-10.664 
N3240 X7.131 Y-10.683 
N3250 X7.156 Y-10.703 
N3260 X7.182 Y-10.724 
N3270 X7.207 Y-10.745 
N3280 X7.231 Y-10.766 
N3290 X7.255 Y-10.788 
N3300 X7.279 Y-10.81 
N3310 X7.302 Y-10.833 
N3320 X7.325 Y-10.856 
N3330 X7.347 Y-10.879 
N3340 X7.369 Y-10.903 
N3350 X7.39 Y-10.928 
N3360 X7.411 Y-10.952 
N3370 X7.432 Y-10.978 
N3380 X7.452 Y-11.003 
N3390 X7.471 Y-11.029 
N3400 X7.49 Y-11.055 
N3410 X7.509 Y-11.082 
N3420 X7.527 Y-11.109 
N3430 X7.545 Y-11.137 
N3440 X7.561 Y-11.164 
N3450 X7.578 Y-11.192 
N3460 X7.594 Y-11.221 
N3470 X7.609 Y-11.25 
N3480 X7.624 Y-11.279 
N3490 X7.638 Y-11.308 
N3500 X7.652 Y-11.338 
N3510 X7.665 Y-11.368 
N3520 X7.678 Y-11.398 
N3530 X7.69 Y-11.429 
N3540 X7.701 Y-11.46 
N3550 X7.712 Y-11.491 
N3560 X7.722 Y-11.523 
N3570 X7.732 Y-11.555 
N3580 X7.74 Y-11.587 
N3590 X7.749 Y-11.619 
N3600 X7.757 Y-11.652 
N3610 X7.764 Y-11.684 
N3620 X7.77 Y-11.717 
N3630 X7.776 Y-11.751 
N3640 X7.781 Y-11.784 
N3650 X7.785 Y-11.818 
N3660 X7.789 Y-11.852 
N3670 X7.792 Y-11.886 
N3680 X7.794 Y-11.921 
N3690 X7.796 Y-11.955 
N3700 X7.797 Y-11.99 
N3710 X7.797 Y-12.008 
N3720 X7.797 Y-12.016 
N3730 X7.797 Y-12.021 
N3740 X7.797 Y-12.027 
N3750 X7.796 Y-12.076 
N3760 X7.794 Y-12.125 
N3770 X7.791 Y-12.173 
N3780 X7.786 Y-12.221 
N3790 X7.779 Y-12.269 
N3800 X7.772 Y-12.316 
N3810 X7.763 Y-12.363 
N3820 X7.753 Y-12.409 
N3830 X7.741 Y-12.455 
N3840 X7.728 Y-12.501 
N3850 X7.714 Y-12.546 
N3860 X7.699 Y-12.59 
N3870 X7.683 Y-12.634 
N3880 X7.666 Y-12.677 
N3890 X7.647 Y-12.72 
N3900 X7.627 Y-12.762 
N3910 X7.606 Y-12.803 
N3920 X7.584 Y-12.844 
N3930 X7.561 Y-12.884 
N3940 X7.537 Y-12.923 
N3950 X7.512 Y-12.962 
N3960 X7.486 Y-13 
N3970 X7.459 Y-13.037 
N3980 X7.431 Y-13.074 
N3990 X7.402 Y-13.109 
N4000 X7.372 Y-13.144 
N4010 X7.341 Y-13.178 
N4020 X7.31 Y-13.211 
N4030 X7.277 Y-13.244 
N4040 X7.244 Y-13.275 
N4050 X7.209 Y-13.306 
N4060 X7.174 Y-13.335 
N4070 X7.138 Y-13.364 
N4080 X7.101 Y-13.392 
N4090 X7.064 Y-13.418 
N4100 X7.026 Y-13.444 
N4110 X6.987 Y-13.469 
N4120 X6.947 Y-13.493 
N4130 X6.907 Y-13.515 
N4140 X6.866 Y-13.537 
N4150 X6.824 Y-13.557 
N4160 X6.782 Y-13.577 
N4170 X6.739 Y-13.595 
N4180 X6.696 Y-13.612 
N4190 X6.652 Y-13.628 
N4200 X6.607 Y-13.643 
N4210 X6.562 Y-13.656 
N4220 X6.517 Y-13.668 
N4230 X6.471 Y-13.679 
N4240 X6.424 Y-13.689 
N4250 X6.377 Y-13.698 
N4260 X6.33 Y-13.705 
N4270 X6.282 Y-13.711 
N4280 X6.234 Y-13.715 
N4290 X6.185 Y-13.719 
N4300 X6.136 Y-13.72 
N4310 X6.087 Y-13.721 
N4320 X6.038 Y-13.72 
N4330 X5.989 Y-13.717 
N4340 X5.94 Y-13.714 
N4350 X5.892 Y-13.708 
N4360 X5.845 Y-13.702 
N4370 X5.797 Y-13.694 
N4380 X5.751 Y-13.685 
N4390 X5.704 Y-13.675 
N4400 X5.658 Y-13.663 
N4410 X5.613 Y-13.65 
N4420 X5.568 Y-13.636 
N4430 X5.524 Y-13.621 
N4440 X5.48 Y-13.605 
N4450 X5.437 Y-13.587 
N4460 X5.394 Y-13.568 
N4470 X5.352 Y-13.548 
N4480 X5.311 Y-13.527 
N4490 X5.27 Y-13.505 
N4500 X5.23 Y-13.482 
N4510 X5.191 Y-13.458 
N4520 X5.153 Y-13.433 
N4530 X5.115 Y-13.407 
N4540 X5.078 Y-13.379 
N4550 X5.041 Y-13.351 
N4560 X5.006 Y-13.322 
N4570 X4.971 Y-13.292 
N4580 X4.937 Y-13.261 
N4590 X4.904 Y-13.229 
N4600 X4.872 Y-13.197 
N4610 X4.84 Y-13.163 
N4620 X4.81 Y-13.129 
N4630 X4.78 Y-13.094 
N4640 X4.752 Y-13.058 
N4650 X4.724 Y-13.021 
N4660 X4.698 Y-12.983 
N4670 X4.672 Y-12.945 
N4680 X4.647 Y-12.906 
N4690 X4.624 Y-12.866 
N4700 X4.601 Y-12.826 
N4710 X4.58 Y-12.785 
N4720 X4.559 Y-12.743 
N4730 X4.54 Y-12.701 
N4740 X4.522 Y-12.658 
N4750 X4.505 Y-12.614 
N4760 X4.489 Y-12.57 
N4770 X4.475 Y-12.526 
N4780 X4.461 Y-12.481 
N4790 X4.449 Y-12.435 
N4800 X4.438 Y-12.389 
N4810 X4.429 Y-12.342 
N4820 X4.42 Y-12.295 
N4830 X4.413 Y-12.248 
N4840 X4.407 Y-12.2 
N4850 X4.403 Y-12.152 
N4860 X4.4 Y-12.103 
N4870 X4.398 Y-12.054 
N4880 X4.398 Y-12.029 
N4890 X4.398 Y-12.023 
N4900 X4.398 Y-12.02 
N4910 X4.398 Y-12.018 
N4920 X4.398 Y-12.009 
N4930 X4.399 Y-11.975 
N4940 X4.4 Y-11.94 
N4950 X4.402 Y-11.905 
N4960 X4.405 Y-11.871 
N4970 X4.408 Y-11.837 
N4980 X4.412 Y-11.803 
N4990 X4.417 Y-11.769 
N5000 X4.422 Y-11.736 
N5010 X4.428 Y-11.703 
N5020 X4.435 Y-11.67 
N5030 X4.442 Y-11.637 
N5040 X4.45 Y-11.605 
N5050 X4.459 Y-11.572 
N5060 X4.468 Y-11.54 
N5070 X4.478 Y-11.509 
N5080 X4.488 Y-11.477 
N5090 X4.499 Y-11.446 
N5100 X4.511 Y-11.415 
N5110 X4.523 Y-11.385 
N5120 X4.536 Y-11.355 
N5130 X4.549 Y-11.325 
N5140 X4.563 Y-11.295 
N5150 X4.578 Y-11.266 
N5160 X4.593 Y-11.237 
N5170 X4.609 Y-11.208 
N5180 X4.625 Y-11.18 
N5190 X4.641 Y-11.152 
N5200 X4.659 Y-11.124 
N5210 X4.676 Y-11.097 
N5220 X4.695 Y-11.07 
N5230 X4.713 Y-11.044 
N5240 X4.733 Y-11.018 
N5250 X4.752 Y-10.992 
N5260 X4.773 Y-10.966 
N5270 X4.793 Y-10.941 
N5280 X4.814 Y-10.917 
N5290 X4.836 Y-10.893 
N5300 X4.858 Y-10.869 
N5310 X4.881 Y-10.846 
N5320 X4.904 Y-10.823 
N5330 X4.927 Y-10.8 
N5340 X4.951 Y-10.778 
N5350 X4.975 Y-10.756 
N5360 X5 Y-10.735 
N5370 X5.025 Y-10.715 
N5380 X5.05 Y-10.694 
N5390 X5.076 Y-10.675 
N5400 X5.103 Y-10.655 
N5410 X5.129 Y-10.636 
N5420 X5.156 Y-10.618 
N5430 X5.184 Y-10.6 
N5440 X5.211 Y-10.583 
N5450 X5.24 Y-10.566 
N5460 X5.268 Y-10.55 
N5470 X5.297 Y-10.534 
N5480 X5.326 Y-10.519 
N5490 X5.341 Y-10.511 
N5500 X5.342 Y-10.51 
N5510 Y-10.508 
N5520 Y-10.504 
N5530 Y-10.5 
N5540 Y-10.494 
N5550 Y-10.486 
N5560 Y-10.478 
N5570 Y-10.468 
N5580 Y-10.456 
N5590 Y-10.444 
N5600 Y-10.43 
N5610 Y-10.416 
N5620 Y-10.4 
N5630 Y-10.383 
N5640 Y-10.365 
N5650 Y-10.346 
N5660 Y-10.325 
N5670 Y-10.304 
N5680 Y-10.282 
N5690 Y-10.259 
N5700 Y-10.235 
N5710 Y-10.21 
N5720 Y-10.184 
N5730 Y-10.157 
N5740 Y-10.13 
N5750 Y-10.101 
N5760 Y-10.072 
N5770 Y-10.042 
N5780 Y-10.012 
N5790 Y-9.98 
N5800 Y-9.948 
N5810 Y-9.915 
N5820 Y-9.882 
N5830 Y-9.848 
N5840 Y-9.814 
N5850 Y-9.779 
N5860 Y-9.743 
N5870 Y-9.707 
N5880 Y-9.67 
N5890 Y-9.596 
N5900 Y-9.519 
N5910 Y-9.442 
N5920 Y-9.363 
N5930 Y-9.283 
N5940 Y-9.203 
N5950 Y-9.121 
N5960 Y-8.958 
N5970 Y-8.795 
N5980 Y-8.713 
N5990 Y-8.633 
N6000 Y-8.553 
N6010 Y-8.474 
N6020 Y-8.397 
N6030 Y-8.32 
N6040 Y-8.246 
N6050 Y-8.209 
N6060 Y-8.173 
N6070 Y-8.138 
N6080 Y-8.102 
N6090 Y-8.068 
N6100 Y-8.034 
N6110 Y-8.001 
N6120 Y-7.968 
N6130 Y-7.936 
N6140 Y-7.905 
N6150 Y-7.874 
N6160 Y-7.844 
N6170 Y-7.815 
N6180 Y-7.786 
N6190 Y-7.759 
N6200 Y-7.732 
N6210 Y-7.706 
N6220 Y-7.681 
N6230 Y-7.657 
N6240 Y-7.634 
N6250 Y-7.612 
N6260 Y-7.591 
N6270 Y-7.57 
N6280 Y-7.551 
N6290 Y-7.533 
N6300 Y-7.516 
N6310 Y-7.5 
N6320 Y-7.486 
N6330 Y-7.472 
N6340 Y-7.46 
N6350 Y-7.448 
N6360 Y-7.438 
N6370 Y-7.43 
N6380 Y-7.422 
N6390 Y-7.416 
N6400 Y-7.412 
N6410 Y-7.408 
N6420 Y-7.406 
N6430 X5.342 Y-7.405 
N6440 X5.341 Y-7.405 
N6450 X5.34 Y-7.403 
N6460 X5.338 Y-7.402 
N6470 X5.336 Y-7.4 
N6480 X5.334 Y-7.397 
N6490 X5.331 Y-7.394 
N6500 X5.328 Y-7.391 
N6510 X5.324 Y-7.387 
N6520 X5.32 Y-7.383 
N6530 X5.315 Y-7.379 
N6540 X5.31 Y-7.374 
N6550 X5.305 Y-7.368 
N6560 X5.299 Y-7.362 
N6570 X5.293 Y-7.356 
N6580 X5.286 Y-7.35 
N6590 X5.279 Y-7.343 
N6600 X5.272 Y-7.336 
N6610 X5.265 Y-7.328 
N6620 X5.256 Y-7.32 
N6630 X5.248 Y-7.311 
N6640 X5.239 Y-7.303 
N6650 X5.23 Y-7.294 
N6660 X5.221 Y-7.284 
N6670 X5.211 Y-7.274 
N6680 X5.201 Y-7.264 
N6690 X5.19 Y-7.253 
N6700 X5.179 Y-7.243 
N6710 X5.168 Y-7.231 
N6720 X5.157 Y-7.22 
N6730 X5.145 Y-7.208 
N6740 X5.132 Y-7.196 
N6750 X5.12 Y-7.183 
N6760 X5.107 Y-7.17 
N6770 X5.081 Y-7.144 
N6780 X5.053 Y-7.116 
N6790 X5.024 Y-7.087 
N6800 X4.994 Y-7.057 
N6810 X4.962 Y-7.026 
N6820 X4.93 Y-6.993 
N6830 X4.897 Y-6.96 
N6840 X4.862 Y-6.926 
N6850 X4.827 Y-6.89 
N6860 X4.79 Y-6.854 
N6870 X4.753 Y-6.816 
N6880 X4.715 Y-6.778 
N6890 X4.676 Y-6.739 
N6900 X4.636 Y-6.699 
N6910 X4.595 Y-6.658 
N6920 X4.553 Y-6.617 
N6930 X4.511 Y-6.574 
N6940 X4.468 Y-6.531 
N6950 X4.424 Y-6.488 
N6960 X4.38 Y-6.443 
N6970 X4.335 Y-6.399 
N6980 X4.29 Y-6.353 
N6990 X4.244 Y-6.307 
N7000 X4.197 Y-6.26 
N7010 X4.15 Y-6.213 
N7020 X4.102 Y-6.166 
N7030 X4.054 Y-6.118 
N7040 X4.006 Y-6.069 
N7050 X3.957 Y-6.02 
N7060 X3.908 Y-5.971 
N7070 X3.809 Y-5.872 
N7080 X3.709 Y-5.772 
N7090 X3.608 Y-5.671 
N7100 X3.506 Y-5.57 
N7110 X3.303 Y-5.367 
N7120 X3.202 Y-5.265 
N7130 X3.101 Y-5.165 
N7140 X3.001 Y-5.065 
N7150 X2.902 Y-4.966 
N7160 X2.854 Y-4.917 
N7170 X2.805 Y-4.868 
N7180 X2.757 Y-4.82 
N7190 X2.709 Y-4.772 
N7200 X2.661 Y-4.725 
N7210 X2.614 Y-4.678 
N7220 X2.568 Y-4.631 
N7230 X2.522 Y-4.586 
N7240 X2.477 Y-4.54 
N7250 X2.432 Y-4.496 
N7260 X2.388 Y-4.452 
N7270 X2.345 Y-4.408 
N7280 X2.302 Y-4.365 
N7290 X2.26 Y-4.324 
N7300 X2.219 Y-4.282 
N7310 X2.179 Y-4.242 
N7320 X2.139 Y-4.202 
N7330 X2.1 Y-4.164 
N7340 X2.062 Y-4.126 
N7350 X2.026 Y-4.089 
N7360 X1.99 Y-4.053 
N7370 X1.955 Y-4.018 
N7380 X1.921 Y-3.984 
N7390 X1.888 Y-3.951 
N7400 X1.856 Y-3.919 
N7410 X1.825 Y-3.888 
N7420 X1.795 Y-3.859 
N7430 X1.767 Y-3.83 
N7440 X1.74 Y-3.803 
N7450 X1.714 Y-3.777 
N7460 X1.701 Y-3.764 
N7470 X1.689 Y-3.752 
N7480 X1.677 Y-3.74 
N7490 X1.665 Y-3.729 
N7500 X1.654 Y-3.717 
N7510 X1.643 Y-3.707 
N7520 X1.633 Y-3.696 
N7530 X1.622 Y-3.686 
N7540 X1.613 Y-3.676 
N7550 X1.603 Y-3.666 
N7560 X1.594 Y-3.657 
N7570 X1.585 Y-3.648 
N7580 X1.577 Y-3.64 
N7590 X1.569 Y-3.632 
N7600 X1.561 Y-3.624 
N7610 X1.553 Y-3.617 
N7620 X1.547 Y-3.61 
N7630 X1.54 Y-3.603 
N7640 X1.534 Y-3.597 
N7650 X1.528 Y-3.591 
N7660 X1.523 Y-3.586 
N7670 X1.518 Y-3.581 
N7680 X1.513 Y-3.576 
N7690 X1.509 Y-3.572 
N7700 X1.505 Y-3.568 
N7710 X1.502 Y-3.565 
N7720 X1.499 Y-3.562 
N7730 X1.496 Y-3.559 
N7740 X1.494 Y-3.557 
N7750 X1.492 Y-3.556 
N7760 X1.491 Y-3.554 
N7770 X1.49 Y-3.554 
N7780 X1.49 Y-3.553 
N7790 X1.488 
N7800 X1.485 
N7810 X1.481 
N7820 X1.476 
N7830 X1.469 
N7840 X1.461 
N7850 X1.452 
N7860 X1.442 
N7870 X1.43 
N7880 X1.418 
N7890 X1.404 
N7900 X1.389 
N7910 X1.373 
N7920 X1.355 
N7930 X1.337 
N7940 X1.317 
N7950 X1.296 
N7960 X1.274 
N7970 X1.252 
N7980 X1.227 
N7990 X1.202 
N8000 X1.176 
N8010 X1.149 
N8020 X1.121 
N8030 X1.091 
N8040 X1.061 
N8050 X1.03 
N8060 X0.998 
N8070 X0.964 
N8080 X0.93 
N8090 X0.895 
N8100 X0.859 
N8110 X0.822 
N8120 X0.784 
N8130 X0.745 
N8140 X0.705 
N8150 X0.665 
N8160 X0.623 
N8170 X0.581 
N8180 X0.537 
N8190 X0.493 
N8200 X0.448 
N8210 X0.403 
N8220 X0.356 
N8230 X0.309 
N8240 X0.261 
N8250 X0.212 
N8260 X0.162 
N8270 X0.112 
N8280 X0.061 
N8290 X0.009 
N8300 X-0.044 
N8310 X-0.097 
N8320 X-0.151 
N8330 X-0.206 
N8340 X-0.261 
N8350 X-0.317 
N8360 X-0.374 
N8370 X-0.431 
N8380 X-0.489 
N8390 X-0.547 
N8400 X-0.606 
N8410 X-0.666 
N8420 X-0.726 
N8430 X-0.787 
N8440 X-0.849 
N8450 X-0.91 
N8460 X-0.973 
N8470 X-1.036 
N8480 X-1.099 
N8490 X-1.163 
N8500 X-1.228 
N8510 X-1.293 
N8520 X-1.358 
N8530 X-1.49 
N8540 X-1.624 
N8550 X-1.759 
N8560 X-1.896 
N8570 X-2.035 
N8580 X-2.174 
N8590 X-2.315 
N8600 X-2.457 
N8610 X-2.6 
N8620 X-2.745 
N8630 X-2.89 
N8640 X-3.035 
N8650 X-3.182 
N8660 X-3.329 
N8670 X-3.625 
N8680 X-3.922 
N8690 X-4.219 
N8700 X-4.516 
N8710 X-4.813 
N8720 X-4.961 
N8730 X-5.108 
N8740 X-5.254 
N8750 X-5.4 
N8760 X-5.545 
N8770 X-5.689 
N8780 X-5.833 
N8790 X-5.975 
N8800 X-6.116 
N8810 X-6.256 
N8820 X-6.394 
N8830 X-6.531 
N8840 X-6.667 
N8850 X-6.801 
N8860 X-6.933 
N8870 X-6.999 
N8880 X-7.064 
N8890 X-7.128 
N8900 X-7.192 
N8910 X-7.256 
N8920 X-7.319 
N8930 X-7.382 
N8940 X-7.444 
N8950 X-7.505 
N8960 X-7.566 
N8970 X-7.626 
N8980 X-7.686 
N8990 X-7.745 
N9000 X-7.804 
N9010 X-7.862 
N9020 X-7.919 
N9030 X-7.976 
N9040 X-8.032 
N9050 X-8.088 
N9060 X-8.143 
N9070 X-8.197 
N9080 X-8.25 
N9090 X-8.303 
N9100 X-8.355 
N9110 X-8.406 
N9120 X-8.457 
N9130 X-8.507 
N9140 X-8.556 
N9150 X-8.604 
N9160 X-8.652 
N9170 X-8.698 
N9180 X-8.744 
N9190 X-8.789 
N9200 X-8.834 
N9210 X-8.877 
N9220 X-8.92 
N9230 X-8.961 
N9240 X-9.002 
N9250 X-9.042 
N9260 X-9.081 
N9270 X-9.119 
N9280 X-9.157 
N9290 X-9.193 
N9300 X-9.228 
N9310 X-9.263 
N9320 X-9.296 
N9330 X-9.329 
N9340 X-9.36 
N9350 X-9.391 
N9360 X-9.42 
N9370 X-9.449 
N9380 X-9.476 
N9390 X-9.503 
N9400 X-9.528 
N9410 X-9.552 
N9420 X-9.575 
N9430 X-9.597 
N9440 X-9.618 
N9450 X-9.638 
N9460 X-9.657 
N9470 X-9.675 
N9480 X-9.691 
N9490 X-9.707 
N9500 X-9.721 
N9510 X-9.734 
N9520 X-9.745 
N9530 X-9.756 
N9540 X-9.765 
N9550 X-9.773 
N9560 X-9.78 
N9570 X-9.786 
N9580 X-9.79 
N9590 X-9.793 
N9600 X-9.795 
N9610 X-9.796 Y-3.553 
N9620 X-9.797 Y-3.552 
N9630 X-9.798 Y-3.551 
N9640 X-9.799 Y-3.55 
N9650 X-9.801 Y-3.548 
N9660 X-9.803 Y-3.546 
N9670 X-9.806 Y-3.543 
N9680 X-9.809 Y-3.54 
N9690 X-9.812 Y-3.537 
N9700 X-9.816 Y-3.533 
N9710 X-9.82 Y-3.529 
N9720 X-9.825 Y-3.524 
N9730 X-9.83 Y-3.519 
N9740 X-9.835 Y-3.514 
N9750 X-9.841 Y-3.508 
N9760 X-9.846 Y-3.502 
N9770 X-9.853 Y-3.496 
N9780 X-9.859 Y-3.489 
N9790 X-9.867 Y-3.482 
N9800 X-9.874 Y-3.475 
N9810 X-9.882 Y-3.467 
N9820 X-9.89 Y-3.459 
N9830 X-9.898 Y-3.451 
N9840 X-9.907 Y-3.442 
N9850 X-9.916 Y-3.433 
N9860 X-9.925 Y-3.424 
N9870 X-9.935 Y-3.414 
N9880 X-9.955 Y-3.394 
N9890 X-9.976 Y-3.373 
N9900 X-9.999 Y-3.35 
N9910 X-10.023 Y-3.326 
N9920 X-10.048 Y-3.301 
N9930 X-10.074 Y-3.275 
N9940 X-10.101 Y-3.248 
N9950 X-10.129 Y-3.22 
N9960 X-10.158 Y-3.191 
N9970 X-10.188 Y-3.161 
N9980 X-10.22 Y-3.129 
N9990 X-10.252 Y-3.097 
N10000 X-10.285 Y-3.064 
N10010 X-10.318 Y-3.03 
N10020 X-10.353 Y-2.996 
N10030 X-10.389 Y-2.96 
N10040 X-10.425 Y-2.924 
N10050 X-10.462 Y-2.887 
N10060 X-10.5 Y-2.849 
N10070 X-10.538 Y-2.81 
N10080 X-10.578 Y-2.771 
N10090 X-10.617 Y-2.731 
N10100 X-10.658 Y-2.691 
N10110 X-10.699 Y-2.65 
N10120 X-10.74 Y-2.608 
N10130 X-10.783 Y-2.566 
N10140 X-10.825 Y-2.524 
N10150 X-10.868 Y-2.481 
N10160 X-10.912 Y-2.437 
N10170 X-10.956 Y-2.393 
N10180 X-11 Y-2.349 
N10190 X-11.045 Y-2.304 
N10200 X-11.135 Y-2.214 
N10210 X-11.227 Y-2.122 
N10220 X-11.319 Y-2.03 
N10230 X-11.412 Y-1.937 
N10240 X-11.505 Y-1.844 
N10250 X-11.692 Y-1.657 
N10260 X-11.785 Y-1.564 
N10270 X-11.877 Y-1.472 
N10280 X-11.969 Y-1.38 
N10290 X-12.059 Y-1.289 
N10300 X-12.104 Y-1.245 
N10310 X-12.149 Y-1.2 
N10320 X-12.193 Y-1.156 
N10330 X-12.237 Y-1.112 
N10340 X-12.28 Y-1.069 
N10350 X-12.323 Y-1.026 
N10360 X-12.366 Y-0.983 
N10370 X-12.408 Y-0.941 
N10380 X-12.449 Y-0.9 
N10390 X-12.49 Y-0.859 
N10400 X-12.53 Y-0.819 
N10410 X-12.57 Y-0.779 
N10420 X-12.609 Y-0.74 
N10430 X-12.647 Y-0.702 
N10440 X-12.685 Y-0.664 
N10450 X-12.721 Y-0.627 
N10460 X-12.757 Y-0.591 
N10470 X-12.793 Y-0.556 
N10480 X-12.827 Y-0.522 
N10490 X-12.861 Y-0.488 
N10500 X-12.893 Y-0.456 
N10510 X-12.925 Y-0.424 
N10520 X-12.956 Y-0.393 
N10530 X-12.986 Y-0.363 
N10540 X-13.015 Y-0.334 
N10550 X-13.043 Y-0.306 
N10560 X-13.069 Y-0.28 
N10570 X-13.095 Y-0.254 
N10580 X-13.12 Y-0.229 
N10590 X-13.143 Y-0.206 
N10600 X-13.165 Y-0.184 
N10610 X-13.186 Y-0.163 
N10620 X-13.206 Y-0.143 
N10630 X-13.216 Y-0.133 
N10640 X-13.225 Y-0.124 
N10650 X-13.233 Y-0.115 
N10660 X-13.242 Y-0.107 
N10670 X-13.25 Y-0.099 
N10680 X-13.258 Y-0.091 
N10690 X-13.265 Y-0.084 
N10700 X-13.272 Y-0.076 
N10710 X-13.279 Y-0.07 
N10720 X-13.286 Y-0.063 
N10730 X-13.292 Y-0.057 
N10740 X-13.298 Y-0.051 
N10750 X-13.303 Y-0.046 
N10760 X-13.308 Y-0.041 
N10770 X-13.313 Y-0.036 
N10780 X-13.317 Y-0.032 
N10790 X-13.321 Y-0.028 
N10800 X-13.324 Y-0.025 
N10810 X-13.327 Y-0.022 
N10820 X-13.33 Y-0.019 
N10830 X-13.333 Y-0.016 
N10840 X-13.335 Y-0.014 
N10850 X-13.336 Y-0.013 
N10860 X-13.337 Y-0.012 
N10870 X-13.338 Y-0.011 
N10880 X-13.338 Y-0.01 
N10890 X-13.339 Y-0.01 
N10900 Y-0.008 
N10910 Y-0.004 
N10920 Y0.002 
N10930 Y0.009 
N10940 Y0.018 
N10950 Y0.028 
N10960 Y0.04 
N10970 Y0.053 
N10980 Y0.068 
N10990 Y0.084 
N11000 Y0.102 
N11010 Y0.121 
N11020 Y0.142 
N11030 Y0.164 
N11040 Y0.187 
N11050 Y0.211 
N11060 Y0.236 
N11070 Y0.263 
N11080 Y0.291 
N11090 Y0.32 
N11100 Y0.35 
N11110 Y0.382 
N11120 Y0.414 
N11130 Y0.447 
N11140 Y0.481 
N11150 Y0.517 
N11160 Y0.553 
N11170 Y0.59 
N11180 Y0.628 
N11190 Y0.666 
N11200 Y0.706 
N11210 Y0.746 
N11220 Y0.787 
N11230 Y0.829 
N11240 Y0.872 
N11250 Y0.915 
N11260 Y0.958 
N11270 Y1.003 
N11280 Y1.048 
N11290 Y1.093 
N11300 Y1.139 
N11310 Y1.232 
N11320 Y1.326 
N11330 Y1.423 
N11340 Y1.52 
N11350 Y1.618 
N11360 Y1.716 
N11370 Y1.915 
N11380 Y2.112 
N11390 Y2.211 
N11400 Y2.308 
N11410 Y2.404 
N11420 Y2.499 
N11430 Y2.592 
N11440 Y2.638 
N11450 Y2.684 
N11460 Y2.728 
N11470 Y2.773 
N11480 Y2.817 
N11490 Y2.86 
N11500 Y2.903 
N11510 Y2.944 
N11520 Y2.986 
N11530 Y3.026 
N11540 Y3.066 
N11550 Y3.105 
N11560 Y3.143 
N11570 Y3.18 
N11580 Y3.216 
N11590 Y3.252 
N11600 Y3.286 
N11610 Y3.32 
N11620 Y3.352 
N11630 Y3.384 
N11640 Y3.414 
N11650 Y3.444 
N11660 Y3.472 
N11670 Y3.499 
N11680 Y3.525 
N11690 Y3.549 
N11700 Y3.573 
N11710 Y3.595 
N11720 Y3.615 
N11730 Y3.635 
N11740 Y3.653 
N11750 Y3.669 
N11760 Y3.685 
N11770 Y3.698 
N11780 Y3.71 
N11790 Y3.721 
N11800 Y3.73 
N11810 Y3.738 
N11820 Y3.744 
N11830 Y3.748 
N11840 Y3.751 
N11850 X-13.368 Y3.766 
N11860 X-13.397 Y3.782 
N11870 X-13.425 Y3.798 
N11880 X-13.454 Y3.815 
N11890 X-13.482 Y3.832 
N11900 X-13.509 Y3.849 
N11910 X-13.537 Y3.867 
N11920 X-13.563 Y3.886 
N11930 X-13.59 Y3.905 
N11940 X-13.616 Y3.924 
N11950 X-13.642 Y3.944 
N11960 X-13.667 Y3.965 
N11970 X-13.692 Y3.986 
N11980 X-13.717 Y4.007 
N11990 X-13.741 Y4.029 
N12000 X-13.764 Y4.051 
N12010 X-13.787 Y4.074 
N12020 X-13.81 Y4.097 
N12030 X-13.833 Y4.121 
N12040 X-13.854 Y4.144 
N12050 X-13.876 Y4.169 
N12060 X-13.897 Y4.194 
N12070 X-13.917 Y4.219 
N12080 X-13.937 Y4.244 
N12090 X-13.957 Y4.27 
N12100 X-13.976 Y4.297 
N12110 X-13.994 Y4.323 
N12120 X-14.012 Y4.35 
N12130 X-14.03 Y4.378 
N12140 X-14.047 Y4.405 
N12150 X-14.063 Y4.434 
N12160 X-14.079 Y4.462 
N12170 X-14.095 Y4.491 
N12180 X-14.109 Y4.52 
N12190 X-14.124 Y4.549 
N12200 X-14.137 Y4.579 
N12210 X-14.151 Y4.609 
N12220 X-14.163 Y4.639 
N12230 X-14.175 Y4.67 
N12240 X-14.186 Y4.701 
N12250 X-14.197 Y4.732 
N12260 X-14.207 Y4.764 
N12270 X-14.217 Y4.796 
N12280 X-14.226 Y4.828 
N12290 X-14.234 Y4.86 
N12300 X-14.242 Y4.893 
N12310 X-14.249 Y4.925 
N12320 X-14.255 Y4.959 
N12330 X-14.261 Y4.992 
N12340 X-14.266 Y5.025 
N12350 X-14.271 Y5.059 
N12360 X-14.274 Y5.093 
N12370 X-14.277 Y5.127 
N12380 X-14.28 Y5.162 
N12390 X-14.282 Y5.196 
N12400 X-14.282 Y5.231 
N12410 X-14.283 Y5.249 
N12420 X-14.283 Y5.257 
N12430 X-14.283 Y5.262 
N12440 X-14.283 Y5.268 
N12450 X-14.282 Y5.317 
N12460 X-14.28 Y5.366 
N12470 X-14.276 Y5.414 
N12480 X-14.271 Y5.462 
N12490 X-14.265 Y5.51 
N12500 X-14.257 Y5.557 
N12510 X-14.248 Y5.604 
N12520 X-14.238 Y5.651 
N12530 X-14.226 Y5.697 
N12540 X-14.214 Y5.742 
N12550 X-14.2 Y5.787 
N12560 X-14.185 Y5.831 
N12570 X-14.168 Y5.875 
N12580 X-14.151 Y5.918 
N12590 X-14.132 Y5.961 
N12600 X-14.113 Y6.003 
N12610 X-14.092 Y6.044 
N12620 X-14.07 Y6.085 
N12630 X-14.047 Y6.125 
N12640 X-14.023 Y6.164 
N12650 X-13.998 Y6.203 
N12660 X-13.972 Y6.241 
N12670 X-13.945 Y6.278 
N12680 X-13.916 Y6.315 
N12690 X-13.887 Y6.35 
N12700 X-13.858 Y6.385 
N12710 X-13.827 Y6.419 
N12720 X-13.795 Y6.452 
N12730 X-13.762 Y6.485 
N12740 X-13.729 Y6.516 
N12750 X-13.695 Y6.547 
N12760 X-13.659 Y6.576 
N12770 X-13.624 Y6.605 
N12780 X-13.587 Y6.633 
N12790 X-13.549 Y6.66 
N12800 X-13.511 Y6.685 
N12810 X-13.472 Y6.71 
N12820 X-13.433 Y6.734 
N12830 X-13.392 Y6.756 
N12840 X-13.351 Y6.778 
N12850 X-13.31 Y6.798 
N12860 X-13.268 Y6.818 
N12870 X-13.225 Y6.836 
N12880 X-13.181 Y6.853 
N12890 X-13.137 Y6.869 
N12900 X-13.093 Y6.884 
N12910 X-13.048 Y6.897 
N12920 X-13.002 Y6.91 
N12930 X-12.956 Y6.921 
N12940 X-12.91 Y6.93 
N12950 X-12.863 Y6.939 
N12960 X-12.815 Y6.946 
N12970 X-12.767 Y6.952 
N12980 X-12.719 Y6.956 
N12990 X-12.67 Y6.96 
N13000 X-12.621 Y6.961 
N13010 X-12.572 Y6.962 
N13020 X-12.523 Y6.961 
N13030 X-12.474 Y6.958 
N13040 X-12.426 Y6.955 
N13050 X-12.378 Y6.95 
N13060 X-12.33 Y6.943 
N13070 X-12.283 Y6.935 
N13080 X-12.236 Y6.926 
N13090 X-12.19 Y6.916 
N13100 X-12.144 Y6.904 
N13110 X-12.098 Y6.891 
N13120 X-12.054 Y6.877 
N13130 X-12.009 Y6.862 
N13140 X-11.966 Y6.846 
N13150 X-11.922 Y6.828 
N13160 X-11.88 Y6.809 
N13170 X-11.838 Y6.789 
N13180 X-11.797 Y6.768 
N13190 X-11.756 Y6.746 
N13200 X-11.716 Y6.723 
N13210 X-11.677 Y6.699 
N13220 X-11.638 Y6.674 
N13230 X-11.6 Y6.648 
N13240 X-11.563 Y6.621 
N13250 X-11.527 Y6.592 
N13260 X-11.491 Y6.563 
N13270 X-11.456 Y6.533 
N13280 X-11.422 Y6.502 
N13290 X-11.389 Y6.471 
N13300 X-11.357 Y6.438 
N13310 X-11.326 Y6.404 
N13320 X-11.295 Y6.37 
N13330 X-11.266 Y6.335 
N13340 X-11.237 Y6.299 
N13350 X-11.21 Y6.262 
N13360 X-11.183 Y6.224 
N13370 X-11.157 Y6.186 
N13380 X-11.133 Y6.147 
N13390 X-11.109 Y6.107 
N13400 X-11.087 Y6.067 
N13410 X-11.065 Y6.026 
N13420 X-11.045 Y5.984 
N13430 X-11.026 Y5.942 
N13440 X-11.007 Y5.899 
N13450 X-10.99 Y5.856 
N13460 X-10.975 Y5.812 
N13470 X-10.96 Y5.767 
N13480 X-10.947 Y5.722 
N13490 X-10.935 Y5.676 
N13500 X-10.924 Y5.63 
N13510 X-10.914 Y5.583 
N13520 X-10.906 Y5.536 
N13530 X-10.899 Y5.489 
N13540 X-10.893 Y5.441 
N13550 X-10.888 Y5.393 
N13560 X-10.885 Y5.344 
N13570 X-10.884 Y5.295 
N13580 X-10.884 Y5.27 
N13590 X-10.884 Y5.264 
N13600 X-10.884 Y5.262 
N13610 X-10.884 Y5.259 
N13620 X-10.884 Y5.251 
N13630 X-10.884 Y5.216 
N13640 X-10.885 Y5.181 
N13650 X-10.887 Y5.146 
N13660 X-10.89 Y5.112 
N13670 X-10.893 Y5.078 
N13680 X-10.898 Y5.044 
N13690 X-10.902 Y5.01 
N13700 X-10.908 Y4.977 
N13710 X-10.914 Y4.944 
N13720 X-10.92 Y4.911 
N13730 X-10.928 Y4.878 
N13740 X-10.936 Y4.846 
N13750 X-10.944 Y4.813 
N13760 X-10.953 Y4.782 
N13770 X-10.963 Y4.75 
N13780 X-10.974 Y4.718 
N13790 X-10.985 Y4.687 
N13800 X-10.996 Y4.656 
N13810 X-11.009 Y4.626 
N13820 X-11.021 Y4.596 
N13830 X-11.035 Y4.566 
N13840 X-11.049 Y4.536 
N13850 X-11.063 Y4.507 
N13860 X-11.078 Y4.478 
N13870 X-11.094 Y4.449 
N13880 X-11.11 Y4.421 
N13890 X-11.127 Y4.393 
N13900 X-11.144 Y4.365 
N13910 X-11.162 Y4.338 
N13920 X-11.18 Y4.311 
N13930 X-11.199 Y4.285 
N13940 X-11.218 Y4.259 
N13950 X-11.238 Y4.233 
N13960 X-11.258 Y4.208 
N13970 X-11.279 Y4.183 
N13980 X-11.3 Y4.158 
N13990 X-11.321 Y4.134 
N14000 X-11.344 Y4.11 
N14010 X-11.366 Y4.087 
N14020 X-11.389 Y4.064 
N14030 X-11.412 Y4.041 
N14040 X-11.436 Y4.019 
N14050 X-11.461 Y3.998 
N14060 X-11.485 Y3.976 
N14070 X-11.51 Y3.956 
N14080 X-11.536 Y3.935 
N14090 X-11.562 Y3.916 
N14100 X-11.588 Y3.896 
N14110 X-11.615 Y3.878 
N14120 X-11.642 Y3.859 
N14130 X-11.669 Y3.841 
N14140 X-11.697 Y3.824 
N14150 X-11.725 Y3.807 
N14160 X-11.753 Y3.791 
N14170 X-11.782 Y3.775 
N14180 X-11.811 Y3.76 
N14190 X-11.826 Y3.752 
N14200 X-11.828 Y3.751 
N14210 Y3.749 
N14220 Y3.746 
N14230 Y3.741 
N14240 Y3.735 
N14250 Y3.727 
N14260 Y3.718 
N14270 Y3.708 
N14280 Y3.697 
N14290 Y3.685 
N14300 Y3.671 
N14310 Y3.656 
N14320 Y3.64 
N14330 Y3.623 
N14340 Y3.604 
N14350 Y3.585 
N14360 Y3.565 
N14370 Y3.543 
N14380 Y3.521 
N14390 Y3.498 
N14400 Y3.473 
N14410 Y3.448 
N14420 Y3.422 
N14430 Y3.395 
N14440 Y3.367 
N14450 Y3.338 
N14460 Y3.309 
N14470 Y3.279 
N14480 Y3.248 
N14490 Y3.216 
N14500 Y3.184 
N14510 Y3.151 
N14520 Y3.117 
N14530 Y3.083 
N14540 Y3.048 
N14550 Y3.013 
N14560 Y2.977 
N14570 Y2.94 
N14580 Y2.903 
N14590 Y2.828 
N14600 Y2.751 
N14610 Y2.673 
N14620 Y2.593 
N14630 Y2.512 
N14640 Y2.431 
N14650 Y2.349 
N14660 Y2.184 
N14670 Y2.019 
N14680 Y1.937 
N14690 Y1.856 
N14700 Y1.775 
N14710 Y1.695 
N14720 Y1.617 
N14730 Y1.54 
N14740 Y1.465 
N14750 Y1.428 
N14760 Y1.391 
N14770 Y1.356 
N14780 Y1.32 
N14790 Y1.285 
N14800 Y1.251 
N14810 Y1.217 
N14820 Y1.184 
N14830 Y1.152 
N14840 Y1.12 
N14850 Y1.089 
N14860 Y1.059 
N14870 Y1.03 
N14880 Y1.001 
N14890 Y0.973 
N14900 Y0.946 
N14910 Y0.92 
N14920 Y0.895 
N14930 Y0.87 
N14940 Y0.847 
N14950 Y0.825 
N14960 Y0.803 
N14970 Y0.783 
N14980 Y0.764 
N14990 Y0.745 
N15000 Y0.728 
N15010 Y0.712 
N15020 Y0.697 
N15030 Y0.684 
N15040 Y0.671 
N15050 Y0.66 
N15060 Y0.65 
N15070 Y0.641 
N15080 Y0.633 
N15090 Y0.627 
N15100 Y0.623 
N15110 Y0.619 
N15120 Y0.617 
N15130 X-11.827 Y0.616 
N15140 X-11.825 Y0.614 
N15150 X-11.822 Y0.611 
N15160 X-11.818 Y0.606 
N15170 X-11.812 Y0.601 
N15180 X-11.806 Y0.594 
N15190 X-11.798 Y0.587 
N15200 X-11.789 Y0.578 
N15210 X-11.779 Y0.568 
N15220 X-11.768 Y0.557 
N15230 X-11.757 Y0.545 
N15240 X-11.744 Y0.533 
N15250 X-11.73 Y0.519 
N15260 X-11.715 Y0.504 
N15270 X-11.699 Y0.488 
N15280 X-11.683 Y0.472 
N15290 X-11.665 Y0.454 
N15300 X-11.647 Y0.436 
N15310 X-11.628 Y0.417 
N15320 X-11.608 Y0.397 
N15330 X-11.587 Y0.376 
N15340 X-11.566 Y0.354 
N15350 X-11.543 Y0.332 
N15360 X-11.52 Y0.309 
N15370 X-11.496 Y0.285 
N15380 X-11.472 Y0.261 
N15390 X-11.447 Y0.236 
N15400 X-11.421 Y0.21 
N15410 X-11.395 Y0.183 
N15420 X-11.368 Y0.156 
N15430 X-11.34 Y0.129 
N15440 X-11.312 Y0.101 
N15450 X-11.283 Y0.072 
N15460 X-11.254 Y0.043 
N15470 X-11.224 Y0.013 
N15480 X-11.194 Y-0.017 
N15490 X-11.164 Y-0.048 
N15500 X-11.133 Y-0.079 
N15510 X-11.101 Y-0.11 
N15520 X-11.069 Y-0.142 
N15530 X-11.037 Y-0.174 
N15540 X-11.005 Y-0.207 
N15550 X-10.972 Y-0.239 
N15560 X-10.905 Y-0.306 
N15570 X-10.838 Y-0.374 
N15580 X-10.769 Y-0.442 
N15590 X-10.7 Y-0.511 
N15600 X-10.63 Y-0.581 
N15610 X-10.561 Y-0.651 
N15620 X-10.42 Y-0.791 
N15630 X-10.351 Y-0.861 
N15640 X-10.281 Y-0.93 
N15650 X-10.212 Y-0.999 
N15660 X-10.144 Y-1.067 
N15670 X-10.076 Y-1.135 
N15680 X-10.01 Y-1.201 
N15690 X-9.977 Y-1.234 
N15700 X-9.945 Y-1.266 
N15710 X-9.913 Y-1.298 
N15720 X-9.881 Y-1.33 
N15730 X-9.85 Y-1.361 
N15740 X-9.819 Y-1.392 
N15750 X-9.789 Y-1.422 
N15760 X-9.759 Y-1.452 
N15770 X-9.729 Y-1.482 
N15780 X-9.7 Y-1.511 
N15790 X-9.672 Y-1.539 
N15800 X-9.644 Y-1.567 
N15810 X-9.617 Y-1.594 
N15820 X-9.59 Y-1.621 
N15830 X-9.564 Y-1.647 
N15840 X-9.538 Y-1.673 
N15850 X-9.514 Y-1.698 
N15860 X-9.489 Y-1.722 
N15870 X-9.466 Y-1.745 
N15880 X-9.443 Y-1.768 
N15890 X-9.421 Y-1.79 
N15900 X-9.4 Y-1.811 
N15910 X-9.38 Y-1.832 
N15920 X-9.36 Y-1.851 
N15930 X-9.341 Y-1.87 
N15940 X-9.323 Y-1.888 
N15950 X-9.306 Y-1.905 
N15960 X-9.29 Y-1.921 
N15970 X-9.275 Y-1.937 
N15980 X-9.26 Y-1.951 
N15990 X-9.247 Y-1.964 
N16000 X-9.234 Y-1.977 
N16010 X-9.223 Y-1.988 
N16020 X-9.213 Y-1.998 
N16030 X-9.203 Y-2.008 
N16040 X-9.195 Y-2.016 
N16050 X-9.188 Y-2.023 
N16060 X-9.182 Y-2.029 
N16070 X-9.177 Y-2.034 
N16080 X-9.173 Y-2.038 
N16090 X-9.17 Y-2.041 
N16100 X-9.169 Y-2.042 
N16110 X-9.168 Y-2.042 
N16120 X-9.167 
N16130 X-9.164 
N16140 X-9.16 
N16150 X-9.155 
N16160 X-9.148 
N16170 X-9.14 
N16180 X-9.131 
N16190 X-9.121 
N16200 X-9.109 
N16210 X-9.097 
N16220 X-9.083 
N16230 X-9.068 
N16240 X-9.052 
N16250 X-9.034 
N16260 X-9.016 
N16270 X-8.996 
N16280 X-8.975 
N16290 X-8.953 
N16300 X-8.93 
N16310 X-8.906 
N16320 X-8.881 
N16330 X-8.855 
N16340 X-8.828 
N16350 X-8.8 
N16360 X-8.77 
N16370 X-8.74 
N16380 X-8.709 
N16390 X-8.677 
N16400 X-8.643 
N16410 X-8.609 
N16420 X-8.574 
N16430 X-8.538 
N16440 X-8.501 
N16450 X-8.463 
N16460 X-8.424 
N16470 X-8.384 
N16480 X-8.343 
N16490 X-8.302 
N16500 X-8.26 
N16510 X-8.216 
N16520 X-8.172 
N16530 X-8.127 
N16540 X-8.082 
N16550 X-8.035 
N16560 X-7.988 
N16570 X-7.94 
N16580 X-7.891 
N16590 X-7.841 
N16600 X-7.791 
N16610 X-7.739 
N16620 X-7.688 
N16630 X-7.635 
N16640 X-7.582 
N16650 X-7.528 
N16660 X-7.473 
N16670 X-7.418 
N16680 X-7.362 
N16690 X-7.305 
N16700 X-7.248 
N16710 X-7.19 
N16720 X-7.132 
N16730 X-7.072 
N16740 X-7.013 
N16750 X-6.953 
N16760 X-6.892 
N16770 X-6.83 
N16780 X-6.768 
N16790 X-6.706 
N16800 X-6.643 
N16810 X-6.58 
N16820 X-6.516 
N16830 X-6.451 
N16840 X-6.386 
N16850 X-6.321 
N16860 X-6.189 
N16870 X-6.055 
N16880 X-5.92 
N16890 X-5.783 
N16900 X-5.644 
N16910 X-5.505 
N16920 X-5.364 
N16930 X-5.222 
N16940 X-5.078 
N16950 X-4.934 
N16960 X-4.789 
N16970 X-4.644 
N16980 X-4.497 
N16990 X-4.35 
N17000 X-4.054 
N17010 X-3.757 
N17020 X-3.46 
N17030 X-3.163 
N17040 X-2.866 
N17050 X-2.718 
N17060 X-2.571 
N17070 X-2.425 
N17080 X-2.279 
N17090 X-2.134 
N17100 X-1.989 
N17110 X-1.846 
N17120 X-1.704 
N17130 X-1.563 
N17140 X-1.423 
N17150 X-1.285 
N17160 X-1.147 
N17170 X-1.012 
N17180 X-0.878 
N17190 X-0.746 
N17200 X-0.68 
N17210 X-0.615 
N17220 X-0.551 
N17230 X-0.486 
N17240 X-0.423 
N17250 X-0.36 
N17260 X-0.297 
N17270 X-0.235 
N17280 X-0.174 
N17290 X-0.113 
N17300 X-0.052 
N17310 X0.007 
N17320 G00 Z5 
N17330 G00 X-0.003 Y1.274 
N17340 G01 Z-5 F254 
N17350 G01 X-0.115 F1200 
N17360 X-0.226 
N17370 X-0.281 
N17380 X-0.336 
N17390 X-0.39 
N17400 X-0.444 
N17410 X-0.497 
N17420 X-0.55 
N17430 X-0.602 
N17440 X-0.653 
N17450 X-0.705 
N17460 X-0.755 
N17470 X-0.805 
N17480 X-0.854 
N17490 X-0.902 
N17500 X-0.95 
N17510 X-0.997 
N17520 X-1.043 
N17530 X-1.088 
N17540 X-1.132 
N17550 X-1.175 
N17560 X-1.218 
N17570 X-1.259 
N17580 X-1.3 
N17590 X-1.339 
N17600 X-1.377 
N17610 X-1.414 
N17620 X-1.451 
N17630 X-1.485 
N17640 X-1.519 
N17650 X-1.552 
N17660 X-1.567 
N17670 X-1.583 
N17680 X-1.598 
N17690 X-1.613 
N17700 X-1.627 
N17710 X-1.641 
N17720 X-1.655 
N17730 X-1.669 
N17740 X-1.682 
N17750 X-1.694 
N17760 X-1.707 
N17770 X-1.719 
N17780 X-1.73 
N17790 X-1.742 
N17800 X-1.753 
N17810 X-1.763 
N17820 X-1.773 
N17830 X-1.783 
N17840 X-1.793 
N17850 X-1.802 
N17860 X-1.81 
N17870 X-1.819 
N17880 X-1.826 
N17890 X-1.834 
N17900 X-1.841 
N17910 X-1.847 
N17920 X-1.854 
N17930 X-1.859 
N17940 X-1.865 
N17950 X-1.87 
N17960 X-1.874 
N17970 X-1.878 
N17980 X-1.882 
N17990 X-1.885 
N18000 X-1.888 
N18010 X-1.89 
N18020 X-1.892 
N18030 X-1.893 
N18040 X-1.894 
N18050 X-1.895 Y1.273 
N18060 X-1.897 Y1.269 
N18070 X-1.9 Y1.262 
N18080 X-1.914 Y1.235 
N18090 X-1.929 Y1.207 
N18100 X-1.945 Y1.181 
N18110 X-1.96 Y1.154 
N18120 X-1.977 Y1.127 
N18130 X-1.993 Y1.101 
N18140 X-2.011 Y1.076 
N18150 X-2.028 Y1.05 
N18160 X-2.046 Y1.025 
N18170 X-2.065 Y1.001 
N18180 X-2.084 Y0.976 
N18190 X-2.103 Y0.952 
N18200 X-2.123 Y0.929 
N18210 X-2.143 Y0.905 
N18220 X-2.163 Y0.882 
N18230 X-2.184 Y0.86 
N18240 X-2.206 Y0.838 
N18250 X-2.227 Y0.816 
N18260 X-2.25 Y0.795 
N18270 X-2.272 Y0.774 
N18280 X-2.295 Y0.753 
N18290 X-2.318 Y0.733 
N18300 X-2.342 Y0.713 
N18310 X-2.366 Y0.694 
N18320 X-2.39 Y0.675 
N18330 X-2.415 Y0.657 
N18340 X-2.44 Y0.638 
N18350 X-2.465 Y0.621 
N18360 X-2.491 Y0.604 
N18370 X-2.517 Y0.587 
N18380 X-2.543 Y0.571 
N18390 X-2.57 Y0.555 
N18400 X-2.597 Y0.54 
N18410 X-2.624 Y0.525 
N18420 X-2.651 Y0.511 
N18430 X-2.679 Y0.497 
N18440 X-2.707 Y0.484 
N18450 X-2.736 Y0.471 
N18460 X-2.764 Y0.459 
N18470 X-2.793 Y0.447 
N18480 X-2.822 Y0.436 
N18490 X-2.852 Y0.425 
N18500 X-2.881 Y0.415 
N18510 X-2.911 Y0.405 
N18520 X-2.941 Y0.396 
N18530 X-2.972 Y0.388 
N18540 X-3.002 Y0.38 
N18550 X-3.033 Y0.372 
N18560 X-3.064 Y0.366 
N18570 X-3.096 Y0.359 
N18580 X-3.127 Y0.354 
N18590 X-3.159 Y0.349 
N18600 X-3.191 Y0.344 
N18610 X-3.223 Y0.34 
N18620 X-3.255 Y0.337 
N18630 X-3.287 Y0.334 
N18640 X-3.32 Y0.332 
N18650 X-3.353 Y0.331 
N18660 X-3.385 Y0.33 
N18670 X-3.402 Y0.33 
N18680 X-3.41 Y0.33 
N18690 X-3.412 Y0.33 
N18700 X-3.415 Y0.33 
N18710 X-3.421 Y0.33 
N18720 X-3.444 Y0.33 
N18730 X-3.467 Y0.33 
N18740 X-3.49 Y0.331 
N18750 X-3.513 Y0.332 
N18760 X-3.559 Y0.336 
N18770 X-3.605 Y0.34 
N18780 X-3.65 Y0.346 
N18790 X-3.695 Y0.353 
N18800 X-3.739 Y0.361 
N18810 X-3.783 Y0.37 
N18820 X-3.827 Y0.381 
N18830 X-3.87 Y0.392 
N18840 X-3.912 Y0.405 
N18850 X-3.955 Y0.418 
N18860 X-3.996 Y0.433 
N18870 X-4.037 Y0.449 
N18880 X-4.078 Y0.465 
N18890 X-4.118 Y0.483 
N18900 X-4.158 Y0.502 
N18910 X-4.197 Y0.522 
N18920 X-4.235 Y0.543 
N18930 X-4.273 Y0.564 
N18940 X-4.311 Y0.587 
N18950 X-4.347 Y0.61 
N18960 X-4.383 Y0.635 
N18970 X-4.418 Y0.66 
N18980 X-4.453 Y0.686 
N18990 X-4.487 Y0.713 
N19000 X-4.52 Y0.741 
N19010 X-4.553 Y0.77 
N19020 X-4.585 Y0.8 
N19030 X-4.616 Y0.83 
N19040 X-4.646 Y0.861 
N19050 X-4.675 Y0.893 
N19060 X-4.704 Y0.925 
N19070 X-4.732 Y0.959 
N19080 X-4.759 Y0.993 
N19090 X-4.785 Y1.027 
N19100 X-4.81 Y1.063 
N19110 X-4.834 Y1.099 
N19120 X-4.858 Y1.136 
N19130 X-4.88 Y1.173 
N19140 X-4.902 Y1.211 
N19150 X-4.922 Y1.249 
N19160 X-4.942 Y1.289 
N19170 X-4.961 Y1.328 
N19180 X-4.978 Y1.368 
N19190 X-4.995 Y1.409 
N19200 X-5.011 Y1.45 
N19210 X-5.025 Y1.492 
N19220 X-5.039 Y1.534 
N19230 X-5.051 Y1.577 
N19240 X-5.063 Y1.62 
N19250 X-5.073 Y1.664 
N19260 X-5.082 Y1.708 
N19270 X-5.09 Y1.752 
N19280 X-5.097 Y1.797 
N19290 X-5.102 Y1.842 
N19300 X-5.106 Y1.888 
N19310 X-5.11 Y1.934 
N19320 X-5.111 Y1.957 
N19330 X-5.112 Y1.98 
N19340 X-5.112 Y2.003 
N19350 X-5.112 Y2.026 
N19360 X-5.112 Y2.05 
N19370 X-5.112 Y2.073 
N19380 X-5.111 Y2.096 
N19390 X-5.11 Y2.119 
N19400 X-5.107 Y2.165 
N19410 X-5.103 Y2.211 
N19420 X-5.097 Y2.256 
N19430 X-5.091 Y2.301 
N19440 X-5.083 Y2.345 
N19450 X-5.074 Y2.389 
N19460 X-5.064 Y2.433 
N19470 X-5.053 Y2.476 
N19480 X-5.04 Y2.519 
N19490 X-5.027 Y2.561 
N19500 X-5.012 Y2.603 
N19510 X-4.997 Y2.644 
N19520 X-4.98 Y2.685 
N19530 X-4.963 Y2.725 
N19540 X-4.944 Y2.765 
N19550 X-4.925 Y2.804 
N19560 X-4.904 Y2.843 
N19570 X-4.883 Y2.881 
N19580 X-4.86 Y2.918 
N19590 X-4.837 Y2.955 
N19600 X-4.813 Y2.991 
N19610 X-4.788 Y3.027 
N19620 X-4.762 Y3.062 
N19630 X-4.735 Y3.096 
N19640 X-4.707 Y3.129 
N19650 X-4.679 Y3.162 
N19660 X-4.649 Y3.194 
N19670 X-4.619 Y3.225 
N19680 X-4.588 Y3.255 
N19690 X-4.557 Y3.285 
N19700 X-4.524 Y3.314 
N19710 X-4.491 Y3.342 
N19720 X-4.457 Y3.369 
N19730 X-4.423 Y3.395 
N19740 X-4.387 Y3.421 
N19750 X-4.351 Y3.445 
N19760 X-4.315 Y3.469 
N19770 X-4.278 Y3.492 
N19780 X-4.24 Y3.513 
N19790 X-4.202 Y3.534 
N19800 X-4.163 Y3.554 
N19810 X-4.123 Y3.573 
N19820 X-4.083 Y3.591 
N19830 X-4.042 Y3.608 
N19840 X-4.001 Y3.624 
N19850 X-3.959 Y3.638 
N19860 X-3.917 Y3.652 
N19870 X-3.875 Y3.665 
N19880 X-3.832 Y3.676 
N19890 X-3.788 Y3.687 
N19900 X-3.744 Y3.696 
N19910 X-3.7 Y3.704 
N19920 X-3.655 Y3.712 
N19930 X-3.61 Y3.717 
N19940 X-3.565 Y3.722 
N19950 X-3.519 Y3.726 
N19960 X-3.496 Y3.727 
N19970 X-3.473 Y3.728 
N19980 X-3.45 Y3.728 
N19990 X-3.426 Y3.729 
N20000 X-3.415 Y3.729 
N20010 X-3.413 Y3.729 
N20020 X-3.412 
N20030 X-3.41 Y3.729 
N20040 X-3.406 Y3.729 
N20050 X-3.389 Y3.729 
N20060 X-3.356 Y3.728 
N20070 X-3.324 Y3.726 
N20080 X-3.291 Y3.724 
N20090 X-3.259 Y3.722 
N20100 X-3.227 Y3.719 
N20110 X-3.195 Y3.715 
N20120 X-3.163 Y3.71 
N20130 X-3.131 Y3.705 
N20140 X-3.1 Y3.7 
N20150 X-3.069 Y3.694 
N20160 X-3.038 Y3.687 
N20170 X-3.007 Y3.679 
N20180 X-2.976 Y3.672 
N20190 X-2.946 Y3.663 
N20200 X-2.916 Y3.654 
N20210 X-2.886 Y3.645 
N20220 X-2.857 Y3.635 
N20230 X-2.827 Y3.624 
N20240 X-2.798 Y3.613 
N20250 X-2.77 Y3.601 
N20260 X-2.741 Y3.589 
N20270 X-2.713 Y3.576 
N20280 X-2.685 Y3.563 
N20290 X-2.657 Y3.549 
N20300 X-2.63 Y3.535 
N20310 X-2.603 Y3.521 
N20320 X-2.576 Y3.506 
N20330 X-2.55 Y3.49 
N20340 X-2.523 Y3.474 
N20350 X-2.498 Y3.457 
N20360 X-2.472 Y3.441 
N20370 X-2.447 Y3.423 
N20380 X-2.422 Y3.405 
N20390 X-2.398 Y3.387 
N20400 X-2.373 Y3.368 
N20410 X-2.35 Y3.349 
N20420 X-2.326 Y3.33 
N20430 X-2.303 Y3.31 
N20440 X-2.28 Y3.289 
N20450 X-2.258 Y3.269 
N20460 X-2.236 Y3.247 
N20470 X-2.214 Y3.226 
N20480 X-2.193 Y3.204 
N20490 X-2.172 Y3.182 
N20500 X-2.152 Y3.159 
N20510 X-2.132 Y3.136 
N20520 X-2.112 Y3.113 
N20530 X-2.093 Y3.089 
N20540 X-2.074 Y3.065 
N20550 X-2.055 Y3.04 
N20560 X-2.037 Y3.016 
N20570 X-2.02 Y2.991 
N20580 X-2.003 Y2.965 
N20590 X-1.986 Y2.94 
N20600 X-1.97 Y2.914 
N20610 X-1.954 Y2.887 
N20620 X-1.939 Y2.861 
N20630 X-1.924 Y2.834 
N20640 X-1.909 Y2.807 
N20650 X-1.902 Y2.793 
N20660 X-1.902 Y2.792 
N20670 X-1.901 
N20680 X-1.9 
N20690 X-1.898 
N20700 X-1.896 
N20710 X-1.893 
N20720 X-1.889 
N20730 X-1.886 
N20740 X-1.881 
N20750 X-1.876 
N20760 X-1.871 
N20770 X-1.865 
N20780 X-1.859 
N20790 X-1.852 
N20800 X-1.845 
N20810 X-1.837 
N20820 X-1.829 
N20830 X-1.82 
N20840 X-1.811 
N20850 X-1.801 
N20860 X-1.791 
N20870 X-1.781 
N20880 X-1.77 
N20890 X-1.758 
N20900 X-1.747 
N20910 X-1.734 
N20920 X-1.722 
N20930 X-1.709 
N20940 X-1.695 
N20950 X-1.681 
N20960 X-1.667 
N20970 X-1.652 
N20980 X-1.637 
N20990 X-1.622 
N21000 X-1.606 
N21010 X-1.59 
N21020 X-1.573 
N21030 X-1.556 
N21040 X-1.538 
N21050 X-1.521 
N21060 X-1.503 
N21070 X-1.484 
N21080 X-1.465 
N21090 X-1.446 
N21100 X-1.427 
N21110 X-1.407 
N21120 X-1.387 
N21130 X-1.366 
N21140 X-1.345 
N21150 X-1.324 
N21160 X-1.281 
N21170 X-1.236 
N21180 X-1.191 
N21190 X-1.144 
N21200 X-1.096 
N21210 X-1.047 
N21220 X-0.997 
N21230 X-0.946 
N21240 X-0.894 
N21250 X-0.841 
N21260 X-0.787 
N21270 X-0.732 
N21280 X-0.677 
N21290 X-0.62 
N21300 X-0.563 
N21310 X-0.505 
N21320 X-0.447 
N21330 X-0.387 
N21340 X-0.327 
N21350 X-0.267 
N21360 X-0.206 
N21370 X-0.145 
N21380 X-0.083 
N21390 X-0.02 
N21400 X0.043 
N21410 X0.106 
N21420 X0.233 
N21430 X0.362 
N21440 X0.491 
N21450 X0.75 
N21460 X0.88 
N21470 X1.009 
N21480 X1.138 
N21490 X1.265 
N21500 X1.329 
N21510 X1.392 
N21520 X1.454 
N21530 X1.517 
N21540 X1.578 
N21550 X1.64 
N21560 X1.7 
N21570 X1.761 
N21580 X1.82 
N21590 X1.879 
N21600 X1.937 
N21610 X1.995 
N21620 X2.052 
N21630 X2.108 
N21640 X2.163 
N21650 X2.218 
N21660 X2.271 
N21670 X2.324 
N21680 X2.375 
N21690 X2.426 
N21700 X2.476 
N21710 X2.524 
N21720 X2.572 
N21730 X2.618 
N21740 X2.663 
N21750 X2.707 
N21760 X2.75 
N21770 X2.771 
N21780 X2.792 
N21790 X2.812 
N21800 X2.832 
N21810 X2.851 
N21820 X2.87 
N21830 X2.889 
N21840 X2.908 
N21850 X2.926 
N21860 X2.944 
N21870 X2.961 
N21880 X2.978 
N21890 X2.995 
N21900 X3.011 
N21910 X3.027 
N21920 X3.043 
N21930 X3.058 
N21940 X3.073 
N21950 X3.087 
N21960 X3.101 
N21970 X3.115 
N21980 X3.128 
N21990 X3.141 
N22000 X3.153 
N22010 X3.165 
N22020 X3.176 
N22030 X3.187 
N22040 X3.198 
N22050 X3.208 
N22060 X3.218 
N22070 X3.227 
N22080 X3.236 
N22090 X3.244 
N22100 X3.252 
N22110 X3.259 
N22120 X3.266 
N22130 X3.272 
N22140 X3.278 
N22150 X3.284 
N22160 X3.289 
N22170 X3.293 
N22180 X3.297 
N22190 X3.301 
N22200 X3.304 
N22210 X3.306 
N22220 X3.308 
N22230 X3.309 
N22240 X3.31 
N22250 X3.311 Y2.792 
N22260 X3.312 Y2.791 
N22270 X3.313 Y2.79 
N22280 X3.314 Y2.788 
N22290 X3.316 Y2.787 
N22300 X3.318 Y2.785 
N22310 X3.32 Y2.782 
N22320 X3.323 Y2.78 
N22330 X3.326 Y2.777 
N22340 X3.329 Y2.774 
N22350 X3.332 Y2.77 
N22360 X3.336 Y2.766 
N22370 X3.34 Y2.762 
N22380 X3.345 Y2.758 
N22390 X3.349 Y2.753 
N22400 X3.354 Y2.748 
N22410 X3.359 Y2.743 
N22420 X3.365 Y2.738 
N22430 X3.37 Y2.732 
N22440 X3.376 Y2.726 
N22450 X3.383 Y2.72 
N22460 X3.389 Y2.713 
N22470 X3.396 Y2.706 
N22480 X3.403 Y2.699 
N22490 X3.41 Y2.692 
N22500 X3.418 Y2.685 
N22510 X3.426 Y2.677 
N22520 X3.434 Y2.669 
N22530 X3.442 Y2.661 
N22540 X3.45 Y2.652 
N22550 X3.459 Y2.643 
N22560 X3.468 Y2.634 
N22570 X3.477 Y2.625 
N22580 X3.487 Y2.616 
N22590 X3.497 Y2.606 
N22600 X3.506 Y2.596 
N22610 X3.527 Y2.576 
N22620 X3.548 Y2.554 
N22630 X3.57 Y2.532 
N22640 X3.593 Y2.509 
N22650 X3.617 Y2.485 
N22660 X3.642 Y2.461 
N22670 X3.667 Y2.435 
N22680 X3.693 Y2.409 
N22690 X3.72 Y2.382 
N22700 X3.748 Y2.355 
N22710 X3.776 Y2.327 
N22720 X3.805 Y2.298 
N22730 X3.834 Y2.268 
N22740 X3.864 Y2.238 
N22750 X3.895 Y2.208 
N22760 X3.926 Y2.177 
N22770 X3.958 Y2.145 
N22780 X3.99 Y2.112 
N22790 X4.023 Y2.08 
N22800 X4.056 Y2.046 
N22810 X4.09 Y2.013 
N22820 X4.124 Y1.978 
N22830 X4.159 Y1.944 
N22840 X4.194 Y1.909 
N22850 X4.229 Y1.873 
N22860 X4.265 Y1.838 
N22870 X4.301 Y1.802 
N22880 X4.337 Y1.765 
N22890 X4.374 Y1.728 
N22900 X4.411 Y1.691 
N22910 X4.448 Y1.654 
N22920 X4.486 Y1.617 
N22930 X4.561 Y1.541 
N22940 X4.637 Y1.465 
N22950 X4.714 Y1.389 
N22960 X5.022 Y1.081 
N22970 X5.098 Y1.004 
N22980 X5.174 Y0.928 
N22990 X5.25 Y0.853 
N23000 X5.287 Y0.815 
N23010 X5.324 Y0.778 
N23020 X5.361 Y0.741 
N23030 X5.398 Y0.705 
N23040 X5.434 Y0.669 
N23050 X5.47 Y0.633 
N23060 X5.505 Y0.597 
N23070 X5.541 Y0.562 
N23080 X5.575 Y0.527 
N23090 X5.61 Y0.493 
N23100 X5.644 Y0.459 
N23110 X5.677 Y0.425 
N23120 X5.71 Y0.392 
N23130 X5.743 Y0.359 
N23140 X5.775 Y0.327 
N23150 X5.807 Y0.296 
N23160 X5.838 Y0.265 
N23170 X5.868 Y0.234 
N23180 X5.898 Y0.205 
N23190 X5.927 Y0.176 
N23200 X5.955 Y0.147 
N23210 X5.983 Y0.119 
N23220 X6.01 Y0.092 
N23230 X6.037 Y0.066 
N23240 X6.063 Y0.04 
N23250 X6.088 Y0.015 
N23260 X6.112 Y-0.009 
N23270 X6.135 Y-0.033 
N23280 X6.158 Y-0.055 
N23290 X6.18 Y-0.077 
N23300 X6.201 Y-0.098 
N23310 X6.221 Y-0.118 
N23320 X6.23 Y-0.128 
N23330 X6.24 Y-0.137 
N23340 X6.249 Y-0.147 
N23350 X6.258 Y-0.156 
N23360 X6.267 Y-0.164 
N23370 X6.275 Y-0.173 
N23380 X6.284 Y-0.181 
N23390 X6.292 Y-0.189 
N23400 X6.299 Y-0.197 
N23410 X6.307 Y-0.205 
N23420 X6.314 Y-0.212 
N23430 X6.321 Y-0.219 
N23440 X6.328 Y-0.226 
N23450 X6.335 Y-0.232 
N23460 X6.341 Y-0.239 
N23470 X6.347 Y-0.245 
N23480 X6.353 Y-0.25 
N23490 X6.358 Y-0.256 
N23500 X6.363 Y-0.261 
N23510 X6.368 Y-0.266 
N23520 X6.373 Y-0.27 
N23530 X6.377 Y-0.275 
N23540 X6.381 Y-0.279 
N23550 X6.385 Y-0.283 
N23560 X6.389 Y-0.286 
N23570 X6.392 Y-0.289 
N23580 X6.395 Y-0.292 
N23590 X6.397 Y-0.295 
N23600 X6.4 Y-0.297 
N23610 X6.402 Y-0.299 
N23620 X6.403 Y-0.301 
N23630 X6.405 Y-0.302 
N23640 X6.406 Y-0.304 
N23650 X6.407 Y-0.304 
N23660 X6.407 Y-0.305 
N23670 X6.408 Y-0.305 
N23680 X6.409 Y-0.306 
N23690 X6.412 Y-0.309 
N23700 X6.413 Y-0.311 
N23710 X6.414 Y-0.312 
N23720 X6.415 Y-0.312 
N23730 X6.415 Y-0.313 
N23740 X6.415 Y-0.312 
N23750 X6.416 Y-0.312 
N23760 X6.417 Y-0.31 
N23770 X6.42 Y-0.308 
N23780 X6.423 Y-0.305 
N23790 X6.426 Y-0.301 
N23800 X6.431 Y-0.297 
N23810 X6.436 Y-0.292 
N23820 X6.442 Y-0.286 
N23830 X6.448 Y-0.279 
N23840 X6.455 Y-0.272 
N23850 X6.463 Y-0.264 
N23860 X6.472 Y-0.256 
N23870 X6.481 Y-0.247 
N23880 X6.49 Y-0.237 
N23890 X6.5 Y-0.227 
N23900 X6.511 Y-0.216 
N23910 X6.522 Y-0.205 
N23920 X6.534 Y-0.193 
N23930 X6.547 Y-0.181 
N23940 X6.56 Y-0.168 
N23950 X6.573 Y-0.154 
N23960 X6.587 Y-0.141 
N23970 X6.601 Y-0.126 
N23980 X6.616 Y-0.111 
N23990 X6.632 Y-0.096 
N24000 X6.648 Y-0.08 
N24010 X6.664 Y-0.064 
N24020 X6.68 Y-0.047 
N24030 X6.697 Y-0.03 
N24040 X6.715 Y-0.013 
N24050 X6.733 Y0.005 
N24060 X6.751 Y0.023 
N24070 X6.77 Y0.042 
N24080 X6.788 Y0.061 
N24090 X6.808 Y0.08 
N24100 X6.827 Y0.1 
N24110 X6.847 Y0.12 
N24120 X6.867 Y0.14 
N24130 X6.888 Y0.16 
N24140 X6.908 Y0.181 
N24150 X6.929 Y0.202 
N24160 X6.951 Y0.223 
N24170 X6.972 Y0.244 
N24180 X7.015 Y0.288 
N24190 X7.06 Y0.332 
N24200 X7.105 Y0.377 
N24210 X7.15 Y0.422 
N24220 X7.196 Y0.468 
N24230 X7.242 Y0.515 
N24240 X7.428 Y0.701 
N24250 X7.475 Y0.747 
N24260 X7.521 Y0.793 
N24270 X7.567 Y0.839 
N24280 X7.612 Y0.884 
N24290 X7.657 Y0.929 
N24300 X7.701 Y0.973 
N24310 X7.744 Y1.016 
N24320 X7.765 Y1.038 
N24330 X7.786 Y1.059 
N24340 X7.807 Y1.08 
N24350 X7.828 Y1.1 
N24360 X7.848 Y1.12 
N24370 X7.868 Y1.14 
N24380 X7.888 Y1.16 
N24390 X7.907 Y1.179 
N24400 X7.926 Y1.199 
N24410 X7.945 Y1.217 
N24420 X7.963 Y1.236 
N24430 X7.981 Y1.254 
N24440 X7.999 Y1.271 
N24450 X8.016 Y1.288 
N24460 X8.033 Y1.305 
N24470 X8.049 Y1.322 
N24480 X8.065 Y1.338 
N24490 X8.081 Y1.353 
N24500 X8.096 Y1.368 
N24510 X8.11 Y1.383 
N24520 X8.125 Y1.397 
N24530 X8.138 Y1.411 
N24540 X8.151 Y1.424 
N24550 X8.164 Y1.436 
N24560 X8.176 Y1.449 
N24570 X8.188 Y1.46 
N24580 X8.199 Y1.471 
N24590 X8.209 Y1.482 
N24600 X8.219 Y1.491 
N24610 X8.228 Y1.501 
N24620 X8.237 Y1.509 
N24630 X8.245 Y1.517 
N24640 X8.252 Y1.525 
N24650 X8.259 Y1.531 
N24660 X8.265 Y1.537 
N24670 X8.27 Y1.543 
N24680 X8.275 Y1.548 
N24690 X8.279 Y1.552 
N24700 X8.282 Y1.555 
N24710 X8.285 Y1.558 
N24720 X8.287 Y1.559 
N24730 X8.288 Y1.56 
N24740 X8.288 Y1.561 
N24750 Y1.562 
N24760 Y1.563 
N24770 Y1.564 
N24780 Y1.565 
N24790 Y1.567 
N24800 Y1.57 
N24810 Y1.572 
N24820 Y1.575 
N24830 Y1.579 
N24840 Y1.582 
N24850 Y1.586 
N24860 Y1.59 
N24870 Y1.595 
N24880 Y1.605 
N24890 Y1.617 
N24900 Y1.629 
N24910 Y1.643 
N24920 Y1.658 
N24930 Y1.674 
N24940 Y1.691 
N24950 Y1.709 
N24960 Y1.729 
N24970 Y1.749 
N24980 Y1.771 
N24990 Y1.793 
N25000 Y1.817 
N25010 Y1.841 
N25020 Y1.866 
N25030 Y1.893 
N25040 Y1.92 
N25050 Y1.948 
N25060 Y1.976 
N25070 Y2.006 
N25080 Y2.036 
N25090 Y2.068 
N25100 Y2.1 
N25110 Y2.132 
N25120 Y2.165 
N25130 Y2.199 
N25140 Y2.234 
N25150 Y2.269 
N25160 Y2.305 
N25170 Y2.342 
N25180 Y2.379 
N25190 Y2.416 
N25200 Y2.454 
N25210 Y2.493 
N25220 Y2.531 
N25230 Y2.571 
N25240 Y2.611 
N25250 Y2.651 
N25260 Y2.691 
N25270 Y2.732 
N25280 Y2.815 
N25290 Y2.898 
N25300 Y2.983 
N25310 Y3.068 
N25320 Y3.24 
N25330 Y3.412 
N25340 Y3.498 
N25350 Y3.583 
N25360 Y3.668 
N25370 Y3.752 
N25380 Y3.835 
N25390 Y3.876 
N25400 Y3.916 
N25410 Y3.957 
N25420 Y3.997 
N25430 Y4.036 
N25440 Y4.075 
N25450 Y4.114 
N25460 Y4.152 
N25470 Y4.19 
N25480 Y4.227 
N25490 Y4.263 
N25500 Y4.299 
N25510 Y4.335 
N25520 Y4.37 
N25530 Y4.404 
N25540 Y4.438 
N25550 Y4.47 
N25560 Y4.503 
N25570 Y4.534 
N25580 Y4.565 
N25590 Y4.595 
N25600 Y4.624 
N25610 Y4.652 
N25620 Y4.679 
N25630 Y4.706 
N25640 Y4.732 
N25650 Y4.756 
N25660 Y4.78 
N25670 Y4.803 
N25680 Y4.825 
N25690 Y4.845 
N25700 Y4.865 
N25710 Y4.884 
N25720 Y4.901 
N25730 Y4.918 
N25740 Y4.933 
N25750 Y4.947 
N25760 Y4.96 
N25770 Y4.972 
N25780 Y4.983 
N25790 Y4.992 
N25800 Y4.996 
N25810 Y5 
N25820 Y5.004 
N25830 Y5.007 
N25840 Y5.01 
N25850 Y5.012 
N25860 Y5.015 
N25870 Y5.016 
N25880 Y5.018 
N25890 Y5.019 
N25900 Y5.02 
N25910 Y5.021 
N25920 X8.287 Y5.021 
N25930 X8.28 Y5.025 
N25940 X8.253 Y5.039 
N25950 X8.225 Y5.054 
N25960 X8.198 Y5.069 
N25970 X8.172 Y5.085 
N25980 X8.145 Y5.101 
N25990 X8.119 Y5.117 
N26000 X8.093 Y5.134 
N26010 X8.068 Y5.152 
N26020 X8.043 Y5.17 
N26030 X8.018 Y5.188 
N26040 X7.994 Y5.207 
N26050 X7.97 Y5.226 
N26060 X7.946 Y5.245 
N26070 X7.923 Y5.265 
N26080 X7.9 Y5.286 
N26090 X7.877 Y5.307 
N26100 X7.855 Y5.328 
N26110 X7.833 Y5.349 
N26120 X7.812 Y5.371 
N26130 X7.791 Y5.394 
N26140 X7.77 Y5.416 
N26150 X7.75 Y5.439 
N26160 X7.73 Y5.463 
N26170 X7.711 Y5.486 
N26180 X7.692 Y5.51 
N26190 X7.673 Y5.535 
N26200 X7.655 Y5.56 
N26210 X7.638 Y5.585 
N26220 X7.62 Y5.61 
N26230 X7.604 Y5.636 
N26240 X7.587 Y5.662 
N26250 X7.572 Y5.688 
N26260 X7.556 Y5.715 
N26270 X7.542 Y5.742 
N26280 X7.527 Y5.769 
N26290 X7.513 Y5.797 
N26300 X7.5 Y5.825 
N26310 X7.487 Y5.853 
N26320 X7.475 Y5.882 
N26330 X7.463 Y5.91 
N26340 X7.452 Y5.939 
N26350 X7.441 Y5.968 
N26360 X7.431 Y5.998 
N26370 X7.421 Y6.028 
N26380 X7.412 Y6.058 
N26390 X7.403 Y6.088 
N26400 X7.395 Y6.118 
N26410 X7.388 Y6.149 
N26420 X7.381 Y6.18 
N26430 X7.375 Y6.211 
N26440 X7.369 Y6.242 
N26450 X7.364 Y6.274 
N26460 X7.359 Y6.306 
N26470 X7.355 Y6.338 
N26480 X7.352 Y6.37 
N26490 X7.349 Y6.402 
N26500 X7.347 Y6.435 
N26510 X7.345 Y6.467 
N26520 X7.344 Y6.5 
N26530 X7.344 Y6.517 
N26540 X7.344 Y6.525 
N26550 X7.344 Y6.529 
N26560 X7.344 Y6.531 
N26570 X7.344 Y6.534 
N26580 X7.344 Y6.557 
N26590 X7.345 Y6.581 
N26600 X7.346 Y6.604 
N26610 X7.347 Y6.627 
N26620 X7.35 Y6.673 
N26630 X7.354 Y6.718 
N26640 X7.36 Y6.763 
N26650 X7.367 Y6.808 
N26660 X7.375 Y6.853 
N26670 X7.384 Y6.897 
N26680 X7.394 Y6.94 
N26690 X7.405 Y6.983 
N26700 X7.418 Y7.026 
N26710 X7.431 Y7.068 
N26720 X7.446 Y7.11 
N26730 X7.461 Y7.151 
N26740 X7.478 Y7.192 
N26750 X7.496 Y7.232 
N26760 X7.514 Y7.272 
N26770 X7.534 Y7.311 
N26780 X7.555 Y7.35 
N26790 X7.576 Y7.388 
N26800 X7.599 Y7.425 
N26810 X7.622 Y7.462 
N26820 X7.646 Y7.498 
N26830 X7.672 Y7.533 
N26840 X7.698 Y7.568 
N26850 X7.725 Y7.602 
N26860 X7.753 Y7.635 
N26870 X7.781 Y7.668 
N26880 X7.811 Y7.699 
N26890 X7.841 Y7.731 
N26900 X7.872 Y7.761 
N26910 X7.904 Y7.79 
N26920 X7.936 Y7.819 
N26930 X7.969 Y7.847 
N26940 X8.003 Y7.874 
N26950 X8.038 Y7.9 
N26960 X8.073 Y7.926 
N26970 X8.109 Y7.95 
N26980 X8.146 Y7.974 
N26990 X8.183 Y7.996 
N27000 X8.221 Y8.018 
N27010 X8.259 Y8.039 
N27020 X8.299 Y8.058 
N27030 X8.338 Y8.077 
N27040 X8.378 Y8.095 
N27050 X8.419 Y8.112 
N27060 X8.46 Y8.128 
N27070 X8.502 Y8.142 
N27080 X8.544 Y8.156 
N27090 X8.587 Y8.168 
N27100 X8.63 Y8.18 
N27110 X8.673 Y8.19 
N27120 X8.717 Y8.199 
N27130 X8.762 Y8.208 
N27140 X8.806 Y8.214 
N27150 X8.852 Y8.22 
N27160 X8.897 Y8.225 
N27170 X8.943 Y8.228 
N27180 X8.966 Y8.229 
N27190 X8.989 Y8.23 
N27200 X9.012 Y8.231 
N27210 X9.036 Y8.231 
N27220 X9.059 Y8.231 
N27230 X9.082 Y8.231 
N27240 X9.105 Y8.23 
N27250 X9.128 Y8.229 
N27260 X9.174 Y8.226 
N27270 X9.22 Y8.222 
N27280 X9.265 Y8.217 
N27290 X9.31 Y8.21 
N27300 X9.355 Y8.202 
N27310 X9.399 Y8.194 
N27320 X9.442 Y8.184 
N27330 X9.486 Y8.173 
N27340 X9.528 Y8.16 
N27350 X9.571 Y8.147 
N27360 X9.613 Y8.133 
N27370 X9.654 Y8.118 
N27380 X9.695 Y8.101 
N27390 X9.735 Y8.084 
N27400 X9.775 Y8.065 
N27410 X9.814 Y8.046 
N27420 X9.853 Y8.025 
N27430 X9.891 Y8.004 
N27440 X9.929 Y7.982 
N27450 X9.965 Y7.959 
N27460 X10.002 Y7.934 
N27470 X10.037 Y7.909 
N27480 X10.072 Y7.883 
N27490 X10.106 Y7.857 
N27500 X10.14 Y7.829 
N27510 X10.172 Y7.801 
N27520 X10.205 Y7.771 
N27530 X10.236 Y7.741 
N27540 X10.266 Y7.711 
N27550 X10.296 Y7.679 
N27560 X10.325 Y7.647 
N27570 X10.353 Y7.614 
N27580 X10.38 Y7.58 
N27590 X10.407 Y7.545 
N27600 X10.432 Y7.51 
N27610 X10.457 Y7.474 
N27620 X10.481 Y7.438 
N27630 X10.503 Y7.401 
N27640 X10.525 Y7.363 
N27650 X10.546 Y7.325 
N27660 X10.566 Y7.286 
N27670 X10.585 Y7.246 
N27680 X10.603 Y7.206 
N27690 X10.62 Y7.166 
N27700 X10.636 Y7.125 
N27710 X10.651 Y7.083 
N27720 X10.665 Y7.041 
N27730 X10.678 Y6.998 
N27740 X10.69 Y6.955 
N27750 X10.7 Y6.912 
N27760 X10.71 Y6.868 
N27770 X10.718 Y6.824 
N27780 X10.725 Y6.779 
N27790 X10.731 Y6.734 
N27800 X10.736 Y6.689 
N27810 X10.74 Y6.643 
N27820 X10.741 Y6.62 
N27830 X10.742 Y6.597 
N27840 X10.743 Y6.574 
N27850 X10.743 Y6.55 
N27860 X10.743 Y6.539 
N27870 X10.743 Y6.533 
N27880 X10.743 Y6.532 
N27890 Y6.53 
N27900 X10.743 Y6.528 
N27910 X10.743 Y6.512 
N27920 X10.743 Y6.479 
N27930 X10.741 Y6.446 
N27940 X10.739 Y6.414 
N27950 X10.737 Y6.381 
N27960 X10.734 Y6.349 
N27970 X10.73 Y6.317 
N27980 X10.725 Y6.285 
N27990 X10.721 Y6.254 
N28000 X10.715 Y6.222 
N28010 X10.709 Y6.191 
N28020 X10.702 Y6.16 
N28030 X10.695 Y6.129 
N28040 X10.687 Y6.099 
N28050 X10.679 Y6.068 
N28060 X10.67 Y6.038 
N28070 X10.66 Y6.008 
N28080 X10.65 Y5.979 
N28090 X10.64 Y5.95 
N28100 X10.628 Y5.92 
N28110 X10.617 Y5.892 
N28120 X10.605 Y5.863 
N28130 X10.592 Y5.835 
N28140 X10.579 Y5.807 
N28150 X10.565 Y5.779 
N28160 X10.551 Y5.752 
N28170 X10.536 Y5.725 
N28180 X10.521 Y5.698 
N28190 X10.506 Y5.671 
N28200 X10.49 Y5.645 
N28210 X10.473 Y5.619 
N28220 X10.456 Y5.594 
N28230 X10.439 Y5.569 
N28240 X10.421 Y5.544 
N28250 X10.402 Y5.519 
N28260 X10.384 Y5.495 
N28270 X10.364 Y5.471 
N28280 X10.345 Y5.447 
N28290 X10.325 Y5.424 
N28300 X10.304 Y5.402 
N28310 X10.283 Y5.379 
N28320 X10.262 Y5.357 
N28330 X10.24 Y5.335 
N28340 X10.218 Y5.314 
N28350 X10.196 Y5.293 
N28360 X10.173 Y5.273 
N28370 X10.15 Y5.253 
N28380 X10.126 Y5.233 
N28390 X10.102 Y5.213 
N28400 X10.078 Y5.195 
N28410 X10.053 Y5.176 
N28420 X10.029 Y5.158 
N28430 X10.003 Y5.14 
N28440 X9.978 Y5.123 
N28450 X9.952 Y5.107 
N28460 X9.925 Y5.09 
N28470 X9.899 Y5.074 
N28480 X9.872 Y5.059 
N28490 X9.845 Y5.044 
N28500 X9.817 Y5.03 
N28510 X9.803 Y5.023 
N28520 X9.8 Y5.021 
N28530 X9.799 Y5.021 
N28540 X9.799 Y5.02 
N28550 Y5.019 
N28560 Y5.018 
N28570 Y5.016 
N28580 Y5.014 
N28590 Y5.012 
N28600 Y5.009 
N28610 Y5.006 
N28620 Y5.002 
N28630 Y4.998 
N28640 Y4.994 
N28650 Y4.989 
N28660 Y4.984 
N28670 Y4.978 
N28680 Y4.973 
N28690 Y4.966 
N28700 Y4.96 
N28710 Y4.953 
N28720 Y4.945 
N28730 Y4.938 
N28740 Y4.929 
N28750 Y4.921 
N28760 Y4.912 
N28770 Y4.903 
N28780 Y4.894 
N28790 Y4.884 
N28800 Y4.874 
N28810 Y4.863 
N28820 Y4.853 
N28830 Y4.83 
N28840 Y4.807 
N28850 Y4.782 
N28860 Y4.756 
N28870 Y4.728 
N28880 Y4.7 
N28890 Y4.67 
N28900 Y4.64 
N28910 Y4.608 
N28920 Y4.575 
N28930 Y4.542 
N28940 Y4.507 
N28950 Y4.471 
N28960 Y4.435 
N28970 Y4.398 
N28980 Y4.359 
N28990 Y4.32 
N29000 Y4.28 
N29010 Y4.24 
N29020 Y4.198 
N29030 Y4.156 
N29040 Y4.114 
N29050 Y4.07 
N29060 Y4.026 
N29070 Y3.981 
N29080 Y3.936 
N29090 Y3.89 
N29100 Y3.844 
N29110 Y3.797 
N29120 Y3.75 
N29130 Y3.702 
N29140 Y3.654 
N29150 Y3.606 
N29160 Y3.557 
N29170 Y3.458 
N29180 Y3.358 
N29190 Y3.258 
N29200 Y3.157 
N29210 Y2.953 
N29220 Y2.75 
N29230 Y2.649 
N29240 Y2.549 
N29250 Y2.45 
N29260 Y2.401 
N29270 Y2.352 
N29280 Y2.303 
N29290 Y2.255 
N29300 Y2.207 
N29310 Y2.16 
N29320 Y2.113 
N29330 Y2.067 
N29340 Y2.021 
N29350 Y1.976 
N29360 Y1.931 
N29370 Y1.887 
N29380 Y1.843 
N29390 Y1.801 
N29400 Y1.758 
N29410 Y1.717 
N29420 Y1.676 
N29430 Y1.636 
N29440 Y1.597 
N29450 Y1.559 
N29460 Y1.522 
N29470 Y1.485 
N29480 Y1.449 
N29490 Y1.415 
N29500 Y1.381 
N29510 Y1.348 
N29520 Y1.316 
N29530 Y1.286 
N29540 Y1.256 
N29550 Y1.228 
N29560 Y1.2 
N29570 Y1.174 
N29580 Y1.149 
N29590 Y1.125 
N29600 Y1.103 
N29610 Y1.092 
N29620 Y1.082 
N29630 Y1.072 
N29640 Y1.062 
N29650 Y1.052 
N29660 Y1.043 
N29670 Y1.034 
N29680 Y1.026 
N29690 Y1.018 
N29700 Y1.01 
N29710 Y1.003 
N29720 Y0.996 
N29730 Y0.989 
N29740 Y0.983 
N29750 Y0.977 
N29760 Y0.971 
N29770 Y0.966 
N29780 Y0.961 
N29790 Y0.957 
N29800 Y0.953 
N29810 Y0.949 
N29820 Y0.946 
N29830 Y0.943 
N29840 Y0.94 
N29850 Y0.938 
N29860 Y0.936 
N29870 Y0.935 
N29880 Y0.934 
N29890 X9.799 Y0.933 
N29900 X9.798 Y0.933 
N29910 X9.797 Y0.932 
N29920 X9.796 Y0.93 
N29930 X9.794 Y0.929 
N29940 X9.792 Y0.927 
N29950 X9.79 Y0.924 
N29960 X9.787 Y0.922 
N29970 X9.784 Y0.919 
N29980 X9.781 Y0.915 
N29990 X9.777 Y0.912 
N30000 X9.773 Y0.908 
N30010 X9.769 Y0.903 
N30020 X9.764 Y0.899 
N30030 X9.759 Y0.894 
N30040 X9.754 Y0.889 
N30050 X9.748 Y0.883 
N30060 X9.743 Y0.877 
N30070 X9.736 Y0.871 
N30080 X9.73 Y0.865 
N30090 X9.723 Y0.858 
N30100 X9.716 Y0.851 
N30110 X9.709 Y0.844 
N30120 X9.702 Y0.836 
N30130 X9.694 Y0.828 
N30140 X9.686 Y0.82 
N30150 X9.677 Y0.812 
N30160 X9.669 Y0.803 
N30170 X9.66 Y0.794 
N30180 X9.65 Y0.785 
N30190 X9.641 Y0.776 
N30200 X9.631 Y0.766 
N30210 X9.621 Y0.756 
N30220 X9.611 Y0.746 
N30230 X9.601 Y0.735 
N30240 X9.59 Y0.725 
N30250 X9.579 Y0.714 
N30260 X9.568 Y0.703 
N30270 X9.556 Y0.691 
N30280 X9.545 Y0.679 
N30290 X9.533 Y0.668 
N30300 X9.521 Y0.655 
N30310 X9.496 Y0.631 
N30320 X9.47 Y0.605 
N30330 X9.443 Y0.578 
N30340 X9.416 Y0.551 
N30350 X9.388 Y0.522 
N30360 X9.358 Y0.493 
N30370 X9.329 Y0.463 
N30380 X9.298 Y0.433 
N30390 X9.267 Y0.401 
N30400 X9.235 Y0.369 
N30410 X9.202 Y0.337 
N30420 X9.169 Y0.303 
N30430 X9.135 Y0.269 
N30440 X9.1 Y0.235 
N30450 X9.065 Y0.2 
N30460 X9.029 Y0.164 
N30470 X8.993 Y0.128 
N30480 X8.956 Y0.091 
N30490 X8.919 Y0.054 
N30500 X8.881 Y0.016 
N30510 X8.843 Y-0.022 
N30520 X8.804 Y-0.061 
N30530 X8.765 Y-0.1 
N30540 X8.726 Y-0.139 
N30550 X8.686 Y-0.179 
N30560 X8.646 Y-0.219 
N30570 X8.606 Y-0.259 
N30580 X8.565 Y-0.3 
N30590 X8.525 Y-0.341 
N30600 X8.442 Y-0.423 
N30610 X8.359 Y-0.506 
N30620 X8.275 Y-0.59 
N30630 X8.107 Y-0.758 
N30640 X7.939 Y-0.927 
N30650 X7.855 Y-1.01 
N30660 X7.772 Y-1.093 
N30670 X7.69 Y-1.176 
N30680 X7.649 Y-1.217 
N30690 X7.608 Y-1.257 
N30700 X7.568 Y-1.298 
N30710 X7.528 Y-1.338 
N30720 X7.488 Y-1.377 
N30730 X7.449 Y-1.417 
N30740 X7.41 Y-1.456 
N30750 X7.371 Y-1.494 
N30760 X7.333 Y-1.532 
N30770 X7.295 Y-1.57 
N30780 X7.258 Y-1.607 
N30790 X7.221 Y-1.644 
N30800 X7.185 Y-1.68 
N30810 X7.149 Y-1.716 
N30820 X7.114 Y-1.751 
N30830 X7.08 Y-1.786 
N30840 X7.046 Y-1.82 
N30850 X7.012 Y-1.853 
N30860 X6.98 Y-1.886 
N30870 X6.947 Y-1.918 
N30880 X6.916 Y-1.949 
N30890 X6.886 Y-1.98 
N30900 X6.856 Y-2.01 
N30910 X6.827 Y-2.039 
N30920 X6.798 Y-2.067 
N30930 X6.771 Y-2.095 
N30940 X6.744 Y-2.121 
N30950 X6.718 Y-2.147 
N30960 X6.693 Y-2.172 
N30970 X6.681 Y-2.184 
N30980 X6.669 Y-2.196 
N30990 X6.658 Y-2.208 
N31000 X6.646 Y-2.219 
N31010 X6.635 Y-2.23 
N31020 X6.624 Y-2.241 
N31030 X6.613 Y-2.252 
N31040 X6.603 Y-2.262 
N31050 X6.593 Y-2.273 
N31060 X6.583 Y-2.282 
N31070 X6.573 Y-2.292 
N31080 X6.564 Y-2.302 
N31090 X6.554 Y-2.311 
N31100 X6.546 Y-2.32 
N31110 X6.537 Y-2.328 
N31120 X6.529 Y-2.337 
N31130 X6.52 Y-2.345 
N31140 X6.513 Y-2.353 
N31150 X6.505 Y-2.36 
N31160 X6.498 Y-2.367 
N31170 X6.491 Y-2.374 
N31180 X6.484 Y-2.381 
N31190 X6.478 Y-2.388 
N31200 X6.472 Y-2.394 
N31210 X6.466 Y-2.4 
N31220 X6.46 Y-2.405 
N31230 X6.455 Y-2.41 
N31240 X6.45 Y-2.415 
N31250 X6.446 Y-2.42 
N31260 X6.441 Y-2.424 
N31270 X6.437 Y-2.428 
N31280 X6.434 Y-2.432 
N31290 X6.43 Y-2.435 
N31300 X6.427 Y-2.438 
N31310 X6.425 Y-2.441 
N31320 X6.422 Y-2.443 
N31330 X6.42 Y-2.445 
N31340 X6.418 Y-2.447 
N31350 X6.417 Y-2.448 
N31360 X6.416 Y-2.449 
N31370 X6.415 Y-2.45 
N31380 X6.414 Y-2.449 
N31390 X6.413 Y-2.448 
N31400 X6.411 Y-2.446 
N31410 X6.409 Y-2.445 
N31420 X6.407 Y-2.442 
N31430 X6.404 Y-2.44 
N31440 X6.401 Y-2.437 
N31450 X6.398 Y-2.433 
N31460 X6.394 Y-2.43 
N31470 X6.39 Y-2.426 
N31480 X6.386 Y-2.421 
N31490 X6.381 Y-2.416 
N31500 X6.376 Y-2.411 
N31510 X6.371 Y-2.406 
N31520 X6.365 Y-2.4 
N31530 X6.359 Y-2.394 
N31540 X6.352 Y-2.388 
N31550 X6.346 Y-2.381 
N31560 X6.338 Y-2.374 
N31570 X6.331 Y-2.366 
N31580 X6.323 Y-2.359 
N31590 X6.315 Y-2.351 
N31600 X6.307 Y-2.342 
N31610 X6.298 Y-2.334 
N31620 X6.289 Y-2.325 
N31630 X6.28 Y-2.316 
N31640 X6.271 Y-2.306 
N31650 X6.261 Y-2.296 
N31660 X6.251 Y-2.286 
N31670 X6.24 Y-2.276 
N31680 X6.23 Y-2.265 
N31690 X6.219 Y-2.254 
N31700 X6.207 Y-2.243 
N31710 X6.196 Y-2.231 
N31720 X6.184 Y-2.219 
N31730 X6.172 Y-2.207 
N31740 X6.16 Y-2.195 
N31750 X6.147 Y-2.182 
N31760 X6.134 Y-2.17 
N31770 X6.121 Y-2.157 
N31780 X6.108 Y-2.143 
N31790 X6.094 Y-2.13 
N31800 X6.08 Y-2.116 
N31810 X6.066 Y-2.102 
N31820 X6.052 Y-2.087 
N31830 X6.037 Y-2.073 
N31840 X6.023 Y-2.058 
N31850 X6.008 Y-2.043 
N31860 X5.977 Y-2.012 
N31870 X5.945 Y-1.981 
N31880 X5.913 Y-1.948 
N31890 X5.879 Y-1.915 
N31900 X5.845 Y-1.881 
N31910 X5.81 Y-1.846 
N31920 X5.775 Y-1.81 
N31930 X5.738 Y-1.774 
N31940 X5.701 Y-1.737 
N31950 X5.664 Y-1.699 
N31960 X5.625 Y-1.661 
N31970 X5.586 Y-1.622 
N31980 X5.547 Y-1.582 
N31990 X5.506 Y-1.542 
N32000 X5.466 Y-1.501 
N32010 X5.424 Y-1.46 
N32020 X5.383 Y-1.418 
N32030 X5.34 Y-1.376 
N32040 X5.298 Y-1.333 
N32050 X5.255 Y-1.29 
N32060 X5.211 Y-1.246 
N32070 X5.167 Y-1.202 
N32080 X5.123 Y-1.158 
N32090 X5.078 Y-1.114 
N32100 X5.034 Y-1.069 
N32110 X4.988 Y-1.024 
N32120 X4.943 Y-0.978 
N32130 X4.852 Y-0.887 
N32140 X4.76 Y-0.795 
N32150 X4.667 Y-0.703 
N32160 X4.575 Y-0.61 
N32170 X4.389 Y-0.425 
N32180 X4.297 Y-0.333 
N32190 X4.206 Y-0.241 
N32200 X4.115 Y-0.15 
N32210 X4.07 Y-0.105 
N32220 X4.025 Y-0.06 
N32230 X3.98 Y-0.016 
N32240 X3.936 Y0.029 
N32250 X3.892 Y0.072 
N32260 X3.849 Y0.116 
N32270 X3.806 Y0.159 
N32280 X3.763 Y0.202 
N32290 X3.721 Y0.244 
N32300 X3.679 Y0.286 
N32310 X3.638 Y0.327 
N32320 X3.597 Y0.368 
N32330 X3.557 Y0.408 
N32340 X3.517 Y0.447 
N32350 X3.478 Y0.486 
N32360 X3.44 Y0.525 
N32370 X3.402 Y0.562 
N32380 X3.365 Y0.599 
N32390 X3.329 Y0.636 
N32400 X3.293 Y0.671 
N32410 X3.259 Y0.706 
N32420 X3.224 Y0.74 
N32430 X3.191 Y0.773 
N32440 X3.159 Y0.806 
N32450 X3.127 Y0.837 
N32460 X3.097 Y0.868 
N32470 X3.082 Y0.883 
N32480 X3.067 Y0.898 
N32490 X3.052 Y0.912 
N32500 X3.038 Y0.927 
N32510 X3.024 Y0.941 
N32520 X3.01 Y0.955 
N32530 X2.996 Y0.968 
N32540 X2.983 Y0.982 
N32550 X2.97 Y0.995 
N32560 X2.957 Y1.007 
N32570 X2.945 Y1.02 
N32580 X2.932 Y1.032 
N32590 X2.92 Y1.044 
N32600 X2.909 Y1.056 
N32610 X2.897 Y1.068 
N32620 X2.886 Y1.079 
N32630 X2.875 Y1.09 
N32640 X2.864 Y1.1 
N32650 X2.854 Y1.111 
N32660 X2.844 Y1.121 
N32670 X2.834 Y1.131 
N32680 X2.825 Y1.14 
N32690 X2.815 Y1.149 
N32700 X2.806 Y1.158 
N32710 X2.798 Y1.167 
N32720 X2.79 Y1.175 
N32730 X2.782 Y1.183 
N32740 X2.774 Y1.191 
N32750 X2.767 Y1.198 
N32760 X2.76 Y1.205 
N32770 X2.753 Y1.212 
N32780 X2.746 Y1.218 
N32790 X2.74 Y1.224 
N32800 X2.735 Y1.23 
N32810 X2.729 Y1.235 
N32820 X2.724 Y1.24 
N32830 X2.72 Y1.245 
N32840 X2.715 Y1.25 
N32850 X2.711 Y1.254 
N32860 X2.708 Y1.257 
N32870 X2.704 Y1.26 
N32880 X2.701 Y1.263 
N32890 X2.699 Y1.266 
N32900 X2.696 Y1.268 
N32910 X2.695 Y1.27 
N32920 X2.693 Y1.272 
N32930 X2.692 Y1.273 
N32940 X2.691 Y1.273 
N32950 X2.691 Y1.274 
N32960 X2.69 Y1.274 
N32970 X2.689 
N32980 X2.688 
N32990 X2.686 
N33000 X2.684 
N33010 X2.681 
N33020 X2.678 
N33030 X2.674 
N33040 X2.67 
N33050 X2.665 
N33060 X2.66 
N33070 X2.655 
N33080 X2.649 
N33090 X2.643 
N33100 X2.636 
N33110 X2.629 
N33120 X2.621 
N33130 X2.613 
N33140 X2.605 
N33150 X2.596 
N33160 X2.587 
N33170 X2.578 
N33180 X2.568 
N33190 X2.557 
N33200 X2.547 
N33210 X2.536 
N33220 X2.524 
N33230 X2.513 
N33240 X2.5 
N33250 X2.488 
N33260 X2.475 
N33270 X2.462 
N33280 X2.448 
N33290 X2.435 
N33300 X2.42 
N33310 X2.406 
N33320 X2.391 
N33330 X2.376 
N33340 X2.36 
N33350 X2.344 
N33360 X2.312 
N33370 X2.278 
N33380 X2.243 
N33390 X2.207 
N33400 X2.169 
N33410 X2.131 
N33420 X2.091 
N33430 X2.051 
N33440 X2.009 
N33450 X1.967 
N33460 X1.923 
N33470 X1.879 
N33480 X1.834 
N33490 X1.788 
N33500 X1.741 
N33510 X1.693 
N33520 X1.645 
N33530 X1.596 
N33540 X1.546 
N33550 X1.495 
N33560 X1.444 
N33570 X1.392 
N33580 X1.34 
N33590 X1.287 
N33600 X1.234 
N33610 X1.18 
N33620 X1.126 
N33630 X1.071 
N33640 X1.016 
N33650 X0.905 
N33660 X0.793 
N33670 X0.68 
N33680 X0.566 
N33690 X0.452 
N33700 X0.224 
N33710 X0.11 
N33720 X-0.003 
N33730 G00 Z5 
N33740 G00 X-6.252 Y2.431 
N33750 G01 Z-5 F254 
N33760 G01 X-6.26 Y2.392 F1200 
N33770 X-6.269 Y2.353 
N33780 X-6.278 Y2.315 
N33790 X-6.289 Y2.277 
N33800 X-6.3 Y2.24 
N33810 X-6.312 Y2.202 
N33820 X-6.325 Y2.166 
N33830 X-6.339 Y2.129 
N33840 X-6.354 Y2.093 
N33850 X-6.369 Y2.058 
N33860 X-6.385 Y2.022 
N33870 X-6.402 Y1.988 
N33880 X-6.42 Y1.953 
N33890 X-6.438 Y1.92 
N33900 X-6.457 Y1.886 
N33910 X-6.477 Y1.853 
N33920 X-6.498 Y1.821 
N33930 X-6.519 Y1.789 
N33940 X-6.541 Y1.758 
N33950 X-6.564 Y1.727 
N33960 X-6.587 Y1.696 
N33970 X-6.611 Y1.666 
N33980 X-6.636 Y1.637 
N33990 X-6.662 Y1.609 
N34000 X-6.688 Y1.58 
N34010 X-6.714 Y1.553 
N34020 X-6.741 Y1.526 
N34030 X-6.769 Y1.5 
N34040 X-6.797 Y1.474 
N34050 X-6.826 Y1.449 
N34060 X-6.856 Y1.425 
N34070 X-6.886 Y1.401 
N34080 X-6.917 Y1.378 
N34090 X-6.948 Y1.355 
N34100 X-6.979 Y1.334 
N34110 X-7.011 Y1.313 
N34120 X-7.044 Y1.292 
N34130 X-7.077 Y1.273 
N34140 X-7.111 Y1.254 
N34150 X-7.145 Y1.236 
N34160 X-7.179 Y1.218 
N34170 X-7.214 Y1.202 
N34180 X-7.25 Y1.186 
N34190 X-7.286 Y1.171 
N34200 X-7.322 Y1.157 
N34210 X-7.358 Y1.143 
N34220 X-7.395 Y1.131 
N34230 X-7.433 Y1.119 
N34240 X-7.47 Y1.108 
N34250 X-7.508 Y1.098 
N34260 X-7.547 Y1.089 
N34270 X-7.586 Y1.081 
N34280 X-7.625 Y1.073 
N34290 X-7.664 Y1.067 
N34300 X-7.704 Y1.061 
N34310 X-7.744 Y1.057 
N34320 X-7.784 Y1.053 
N34330 X-7.824 Y1.05 
N34340 X-7.865 Y1.048 
N34350 X-7.906 Y1.047 
N34360 X-7.947 Y1.047 
N34370 X-7.988 Y1.048 
N34380 X-8.029 Y1.05 
N34390 X-8.069 Y1.053 
N34400 X-8.109 Y1.057 
N34410 X-8.149 Y1.062 
N34420 X-8.189 Y1.068 
N34430 X-8.228 Y1.075 
N34440 X-8.267 Y1.082 
N34450 X-8.306 Y1.091 
N34460 X-8.344 Y1.1 
N34470 X-8.382 Y1.11 
N34480 X-8.42 Y1.121 
N34490 X-8.457 Y1.133 
N34500 X-8.494 Y1.146 
N34510 X-8.53 Y1.16 
N34520 X-8.566 Y1.174 
N34530 X-8.602 Y1.189 
N34540 X-8.637 Y1.205 
N34550 X-8.672 Y1.222 
N34560 X-8.707 Y1.239 
N34570 X-8.741 Y1.258 
N34580 X-8.774 Y1.277 
N34590 X-8.807 Y1.296 
N34600 X-8.84 Y1.317 
N34610 X-8.872 Y1.338 
N34620 X-8.903 Y1.36 
N34630 X-8.934 Y1.382 
N34640 X-8.965 Y1.406 
N34650 X-8.995 Y1.429 
N34660 X-9.024 Y1.454 
N34670 X-9.053 Y1.479 
N34680 X-9.081 Y1.505 
N34690 X-9.109 Y1.531 
N34700 X-9.136 Y1.558 
N34710 X-9.162 Y1.586 
N34720 X-9.188 Y1.614 
N34730 X-9.214 Y1.643 
N34740 X-9.238 Y1.672 
N34750 X-9.262 Y1.702 
N34760 X-9.285 Y1.733 
N34770 X-9.308 Y1.764 
N34780 X-9.33 Y1.795 
N34790 X-9.351 Y1.827 
N34800 X-9.371 Y1.86 
N34810 X-9.391 Y1.893 
N34820 X-9.41 Y1.926 
N34830 X-9.429 Y1.96 
N34840 X-9.446 Y1.995 
N34850 X-9.463 Y2.029 
N34860 X-9.479 Y2.065 
N34870 X-9.494 Y2.1 
N34880 X-9.509 Y2.136 
N34890 X-9.522 Y2.173 
N34900 X-9.535 Y2.21 
N34910 X-9.547 Y2.247 
N34920 X-9.558 Y2.285 
N34930 X-9.568 Y2.323 
N34940 X-9.578 Y2.361 
N34950 X-9.586 Y2.4 
N34960 X-9.594 Y2.439 
N34970 X-9.601 Y2.478 
N34980 X-9.607 Y2.517 
N34990 X-9.611 Y2.557 
N35000 X-9.615 Y2.597 
N35010 X-9.619 Y2.638 
N35020 X-9.621 Y2.679 
N35030 X-9.622 Y2.719 
N35040 X-9.622 Y2.74 
N35050 X-9.622 Y2.745 
N35060 Y2.747 
N35070 X-9.622 Y2.749 
N35080 X-9.622 Y2.757 
N35090 X-9.622 Y2.786 
N35100 X-9.621 Y2.815 
N35110 X-9.619 Y2.843 
N35120 X-9.617 Y2.872 
N35130 X-9.615 Y2.901 
N35140 X-9.612 Y2.929 
N35150 X-9.609 Y2.957 
N35160 X-9.605 Y2.985 
N35170 X-9.601 Y3.013 
N35180 X-9.596 Y3.041 
N35190 X-9.591 Y3.069 
N35200 X-9.586 Y3.096 
N35210 X-9.579 Y3.124 
N35220 X-9.573 Y3.151 
N35230 X-9.566 Y3.178 
N35240 X-9.559 Y3.204 
N35250 X-9.551 Y3.231 
N35260 X-9.543 Y3.257 
N35270 X-9.534 Y3.284 
N35280 X-9.525 Y3.31 
N35290 X-9.516 Y3.335 
N35300 X-9.506 Y3.361 
N35310 X-9.495 Y3.386 
N35320 X-9.485 Y3.412 
N35330 X-9.474 Y3.437 
N35340 X-9.462 Y3.461 
N35350 X-9.45 Y3.486 
N35360 X-9.438 Y3.51 
N35370 X-9.425 Y3.534 
N35380 X-9.412 Y3.558 
N35390 X-9.399 Y3.582 
N35400 X-9.385 Y3.605 
N35410 X-9.371 Y3.628 
N35420 X-9.357 Y3.651 
N35430 X-9.342 Y3.674 
N35440 X-9.326 Y3.696 
N35450 X-9.311 Y3.718 
N35460 X-9.295 Y3.74 
N35470 X-9.279 Y3.762 
N35480 X-9.262 Y3.783 
N35490 X-9.245 Y3.804 
N35500 X-9.228 Y3.825 
N35510 X-9.21 Y3.846 
N35520 X-9.192 Y3.866 
N35530 X-9.174 Y3.886 
N35540 X-9.156 Y3.906 
N35550 X-9.137 Y3.925 
N35560 X-9.118 Y3.944 
N35570 X-9.098 Y3.963 
N35580 X-9.078 Y3.981 
N35590 X-9.058 Y3.999 
N35600 X-9.038 Y4.017 
N35610 X-9.017 Y4.035 
N35620 X-8.997 Y4.052 
N35630 X-8.975 Y4.069 
N35640 X-8.954 Y4.086 
N35650 X-8.932 Y4.102 
N35660 X-8.91 Y4.118 
N35670 X-8.888 Y4.134 
N35680 X-8.865 Y4.149 
N35690 X-8.842 Y4.164 
N35700 X-8.819 Y4.178 
N35710 X-8.796 Y4.193 
N35720 X-8.773 Y4.206 
N35730 X-8.749 Y4.22 
N35740 X-8.725 Y4.233 
N35750 X-8.701 Y4.246 
N35760 X-8.688 Y4.252 
N35770 X-8.682 Y4.255 
N35780 X-8.679 Y4.257 
N35790 X-8.678 Y4.258 
N35800 Y4.259 
N35810 Y4.26 
N35820 Y4.262 
N35830 Y4.265 
N35840 Y4.268 
N35850 Y4.272 
N35860 Y4.276 
N35870 Y4.281 
N35880 Y4.286 
N35890 Y4.292 
N35900 Y4.298 
N35910 Y4.305 
N35920 Y4.312 
N35930 Y4.32 
N35940 Y4.328 
N35950 Y4.336 
N35960 Y4.345 
N35970 Y4.355 
N35980 Y4.365 
N35990 Y4.375 
N36000 Y4.386 
N36010 Y4.397 
N36020 Y4.408 
N36030 Y4.42 
N36040 Y4.432 
N36050 Y4.445 
N36060 Y4.458 
N36070 Y4.471 
N36080 Y4.484 
N36090 Y4.498 
N36100 Y4.513 
N36110 Y4.542 
N36120 Y4.573 
N36130 Y4.604 
N36140 Y4.637 
N36150 Y4.671 
N36160 Y4.705 
N36170 Y4.741 
N36180 Y4.777 
N36190 Y4.814 
N36200 Y4.851 
N36210 Y4.889 
N36220 Y4.928 
N36230 Y4.967 
N36240 Y5.045 
N36250 Y5.125 
N36260 Y5.285 
N36270 Y5.364 
N36280 Y5.403 
N36290 Y5.441 
N36300 Y5.479 
N36310 Y5.517 
N36320 Y5.554 
N36330 Y5.59 
N36340 Y5.626 
N36350 Y5.66 
N36360 Y5.694 
N36370 Y5.727 
N36380 Y5.759 
N36390 Y5.79 
N36400 Y5.819 
N36410 Y5.833 
N36420 Y5.848 
N36430 Y5.861 
N36440 Y5.875 
N36450 Y5.888 
N36460 Y5.9 
N36470 Y5.912 
N36480 Y5.924 
N36490 Y5.936 
N36500 Y5.947 
N36510 Y5.958 
N36520 Y5.968 
N36530 Y5.978 
N36540 Y5.988 
N36550 Y5.997 
N36560 Y6.006 
N36570 Y6.014 
N36580 Y6.022 
N36590 Y6.029 
N36600 Y6.036 
N36610 Y6.042 
N36620 Y6.048 
N36630 Y6.053 
N36640 Y6.058 
N36650 Y6.063 
N36660 Y6.066 
N36670 Y6.07 
N36680 Y6.073 
N36690 Y6.075 
N36700 Y6.076 
N36710 Y6.078 
N36720 X-8.677 Y6.079 
N36730 X-8.676 Y6.079 
N36740 X-8.676 Y6.08 
N36750 X-8.674 Y6.081 
N36760 X-8.673 Y6.083 
N36770 X-8.671 Y6.085 
N36780 X-8.669 Y6.087 
N36790 X-8.667 Y6.089 
N36800 X-8.665 Y6.091 
N36810 X-8.662 Y6.094 
N36820 X-8.659 Y6.097 
N36830 X-8.656 Y6.1 
N36840 X-8.653 Y6.103 
N36850 X-8.649 Y6.107 
N36860 X-8.646 Y6.11 
N36870 X-8.641 Y6.114 
N36880 X-8.637 Y6.119 
N36890 X-8.633 Y6.123 
N36900 X-8.623 Y6.133 
N36910 X-8.613 Y6.143 
N36920 X-8.602 Y6.154 
N36930 X-8.589 Y6.166 
N36940 X-8.576 Y6.179 
N36950 X-8.563 Y6.193 
N36960 X-8.548 Y6.208 
N36970 X-8.533 Y6.223 
N36980 X-8.517 Y6.239 
N36990 X-8.5 Y6.256 
N37000 X-8.482 Y6.273 
N37010 X-8.464 Y6.292 
N37020 X-8.445 Y6.311 
N37030 X-8.426 Y6.33 
N37040 X-8.405 Y6.351 
N37050 X-8.384 Y6.372 
N37060 X-8.363 Y6.393 
N37070 X-8.34 Y6.415 
N37080 X-8.318 Y6.438 
N37090 X-8.294 Y6.462 
N37100 X-8.27 Y6.486 
N37110 X-8.246 Y6.51 
N37120 X-8.22 Y6.535 
N37130 X-8.195 Y6.561 
N37140 X-8.169 Y6.587 
N37150 X-8.142 Y6.614 
N37160 X-8.115 Y6.641 
N37170 X-8.087 Y6.669 
N37180 X-8.059 Y6.697 
N37190 X-8.03 Y6.725 
N37200 X-8.001 Y6.754 
N37210 X-7.972 Y6.784 
N37220 X-7.942 Y6.814 
N37230 X-7.912 Y6.844 
N37240 X-7.881 Y6.874 
N37250 X-7.85 Y6.905 
N37260 X-7.819 Y6.937 
N37270 X-7.788 Y6.968 
N37280 X-7.756 Y7 
N37290 X-7.724 Y7.032 
N37300 X-7.691 Y7.065 
N37310 X-7.658 Y7.097 
N37320 X-7.625 Y7.13 
N37330 X-7.592 Y7.164 
N37340 X-7.525 Y7.231 
N37350 X-7.457 Y7.299 
N37360 X-7.389 Y7.367 
N37370 X-7.32 Y7.436 
N37380 X-7.25 Y7.505 
N37390 X-7.181 Y7.575 
N37400 X-7.041 Y7.715 
N37410 X-6.902 Y7.854 
N37420 X-6.832 Y7.923 
N37430 X-6.764 Y7.992 
N37440 X-6.695 Y8.061 
N37450 X-6.628 Y8.128 
N37460 X-6.561 Y8.195 
N37470 X-6.528 Y8.228 
N37480 X-6.495 Y8.261 
N37490 X-6.463 Y8.293 
N37500 X-6.43 Y8.326 
N37510 X-6.398 Y8.358 
N37520 X-6.367 Y8.389 
N37530 X-6.335 Y8.421 
N37540 X-6.304 Y8.452 
N37550 X-6.273 Y8.482 
N37560 X-6.243 Y8.513 
N37570 X-6.213 Y8.543 
N37580 X-6.184 Y8.572 
N37590 X-6.155 Y8.601 
N37600 X-6.126 Y8.63 
N37610 X-6.098 Y8.658 
N37620 X-6.07 Y8.686 
N37630 X-6.042 Y8.713 
N37640 X-6.016 Y8.74 
N37650 X-5.989 Y8.767 
N37660 X-5.963 Y8.792 
N37670 X-5.938 Y8.818 
N37680 X-5.913 Y8.843 
N37690 X-5.889 Y8.867 
N37700 X-5.865 Y8.89 
N37710 X-5.842 Y8.913 
N37720 X-5.82 Y8.936 
N37730 X-5.798 Y8.958 
N37740 X-5.777 Y8.979 
N37750 X-5.756 Y8.999 
N37760 X-5.737 Y9.019 
N37770 X-5.717 Y9.038 
N37780 X-5.699 Y9.057 
N37790 X-5.681 Y9.075 
N37800 X-5.664 Y9.092 
N37810 X-5.648 Y9.108 
N37820 X-5.632 Y9.124 
N37830 X-5.617 Y9.138 
N37840 X-5.603 Y9.152 
N37850 X-5.59 Y9.166 
N37860 X-5.578 Y9.178 
N37870 X-5.566 Y9.19 
N37880 X-5.555 Y9.2 
N37890 X-5.546 Y9.21 
N37900 X-5.541 Y9.215 
N37910 X-5.537 Y9.219 
N37920 X-5.532 Y9.223 
N37930 X-5.529 Y9.227 
N37940 X-5.525 Y9.231 
N37950 X-5.521 Y9.235 
N37960 X-5.518 Y9.238 
N37970 X-5.515 Y9.241 
N37980 X-5.512 Y9.244 
N37990 X-5.51 Y9.246 
N38000 X-5.507 Y9.248 
N38010 X-5.505 Y9.251 
N38020 X-5.503 Y9.252 
N38030 X-5.502 Y9.254 
N38040 X-5.501 Y9.255 
N38050 X-5.499 Y9.256 
N38060 X-5.499 Y9.257 
N38070 X-5.498 Y9.258 
N38080 X-5.497 Y9.258 
N38090 X-5.496 
N38100 X-5.494 
N38110 X-5.492 
N38120 X-5.489 
N38130 X-5.485 
N38140 X-5.481 
